C03641=1038.429,245.256,390.466,171.048,41.965,157.999
C03642=1038.436,245.505,390.436,171.051,41.966,157.999
C03643=1038.442,245.753,390.407,171.053,41.968,158.000
C03644=1038.448,246.001,390.378,171.057,41.969,158.001
C03645=1038.454,246.250,390.349,171.059,41.970,158.001
C03646=1038.461,246.497,390.321,171.062,41.972,158.001
C03647=1038.468,246.746,390.291,171.065,41.973,158.002
C03648=1038.474,246.994,390.262,171.068,41.974,158.002
C03649=1038.481,247.242,390.233,171.070,41.976,158.003
C03650=1038.487,247.491,390.204,171.074,41.977,158.003
C03651=1038.494,247.739,390.175,171.077,41.979,158.004
C03652=1038.501,247.987,390.146,171.079,41.980,158.004
C03653=1038.507,248.235,390.117,171.083,41.981,158.005
C03654=1038.515,248.549,390.080,171.085,41.983,158.005
C03655=1038.524,248.863,390.043,171.089,41.985,158.006
C03656=1038.532,249.178,390.007,171.092,41.986,158.006
C03657=1038.541,249.493,389.970,171.096,41.988,158.007
C03658=1038.547,249.741,389.941,171.100,41.989,158.007
C03659=1038.553,249.989,389.912,171.102,41.991,158.008
C03660=1038.560,250.237,389.881,171.105,41.992,158.008
C03661=1038.566,250.485,389.852,171.108,41.994,158.009
C03662=1038.573,250.733,389.823,171.111,41.995,158.009
C03663=1038.579,250.981,389.794,171.114,41.996,158.010
C03664=1038.587,251.230,389.765,171.117,41.998,158.010
C03665=1038.593,251.478,389.736,171.119,41.998,158.011
C03666=1038.600,251.726,389.706,171.123,42.000,158.011
C03667=1038.606,251.974,389.677,171.126,42.001,158.012
C03668=1038.612,252.223,389.648,171.129,42.003,158.012
C03669=1038.619,252.471,389.619,171.132,42.004,158.013
C03670=1038.626,252.719,389.589,171.134,42.005,158.013
C03671=1038.633,252.967,389.561,171.138,42.007,158.014
C03672=1038.640,253.216,389.531,171.140,42.008,158.014
C03673=1038.646,253.463,389.501,171.144,42.009,158.015
C03674=1038.653,253.712,389.472,171.146,42.011,158.015
C03675=1038.659,253.960,389.443,171.149,42.012,158.016
C03676=1038.666,254.208,389.414,171.152,42.013,158.016
C03677=1038.673,254.456,389.384,171.155,42.015,158.016
C03678=1038.679,254.705,389.355,171.159,42.016,158.017
C03679=1038.686,254.953,389.325,171.161,42.018,158.017
C03680=1038.693,255.201,389.296,171.165,42.018,158.018
C03681=1038.700,255.449,389.267,171.167,42.020,158.018
C03682=1038.707,255.697,389.237,171.171,42.021,158.019
C03683=1038.713,255.946,389.208,171.173,42.023,158.019
C03684=1038.720,256.194,389.179,171.176,42.024,158.020
C03685=1038.727,256.442,389.148,171.179,42.025,158.020
C03686=1038.733,256.690,389.119,171.182,42.027,158.021
C03687=1038.740,256.938,389.089,171.186,42.028,158.021
C03688=1038.746,257.187,389.060,171.188,42.029,158.022
C03689=1038.754,257.435,389.030,171.192,42.031,158.022
C03690=1038.761,257.683,389.002,171.194,42.032,158.023
C03691=1038.768,257.931,388.972,171.198,42.033,158.023
C03692=1038.774,258.179,388.943,171.200,42.034,158.024
C03693=1038.781,258.427,388.912,171.204,42.036,158.024
C03694=1038.787,258.675,388.883,171.206,42.037,158.025
C03695=1038.795,258.924,388.853,171.210,42.038,158.025
C03696=1038.801,259.172,388.824,171.212,42.040,158.026
C03697=1038.808,259.420,388.794,171.216,42.041,158.026
C03698=1038.815,259.669,388.765,171.219,42.043,158.027
C03699=1038.821,259.916,388.735,171.222,42.044,158.027
C03700=1038.829,260.164,388.705,171.225,42.045,158.027
C03701=1038.835,260.413,388.676,171.228,42.046,158.028
C03702=1038.843,260.660,388.646,171.232,42.048,158.029
C03703=1038.849,260.909,388.617,171.234,42.049,158.029
C03704=1038.856,261.157,388.587,171.238,42.050,158.029
C03705=1038.863,261.405,388.557,171.240,42.052,158.030
C03706=1038.869,261.653,388.528,171.244,42.053,158.030
C03707=1038.877,261.901,388.498,171.246,42.055,158.031
C03708=1038.884,262.150,388.468,171.250,42.056,158.032
C03709=1038.890,262.397,388.437,171.253,42.058,158.032
C03710=1038.898,262.711,388.400,171.256,42.059,158.033
C03711=1038.906,263.023,388.362,171.261,42.061,158.033
C03712=1038.915,263.336,388.324,171.265,42.063,158.034
C03713=1038.923,263.649,388.287,171.268,42.064,158.034
C03714=1038.930,263.897,388.256,171.272,42.066,158.035
C03715=1038.936,264.145,388.226,171.275,42.067,158.036
C03716=1038.943,264.393,388.196,171.278,42.069,158.036
C03717=1038.950,264.641,388.166,171.281,42.070,158.037
C03718=1038.956,264.889,388.135,171.284,42.072,158.037
C03719=1038.963,265.137,388.105,171.287,42.073,158.038
C03720=1038.971,265.385,388.075,171.291,42.075,158.038
C03721=1038.976,265.633,388.045,171.293,42.076,158.039
C03722=1038.984,265.881,388.015,171.297,42.077,158.039
C03723=1038.991,266.130,387.985,171.300,42.079,158.040
C03724=1038.997,266.378,387.954,171.303,42.080,158.040
C03725=1039.004,266.626,387.924,171.307,42.082,158.041
C03726=1039.011,266.874,387.894,171.309,42.083,158.041
C03727=1039.017,267.122,387.864,171.313,42.085,158.042
C03728=1039.024,267.370,387.834,171.316,42.086,158.042
C03729=1039.031,267.618,387.803,171.319,42.088,158.043
C03730=1039.037,267.866,387.773,171.323,42.089,158.043
C03731=1039.044,268.114,387.743,171.325,42.091,158.044
C03732=1039.050,268.363,387.712,171.329,42.092,158.044
C03733=1039.057,268.610,387.683,171.332,42.093,158.045
C03734=1039.064,268.858,387.651,171.335,42.095,158.045
C03735=1039.071,269.106,387.621,171.339,42.096,158.046
C03736=1039.077,269.354,387.591,171.341,42.098,158.046
C03737=1039.084,269.602,387.560,171.345,42.099,158.047
C03738=1039.090,269.851,387.530,171.348,42.101,158.048
C03739=1039.098,270.099,387.499,171.351,42.102,158.048
C03740=1039.103,270.346,387.469,171.355,42.104,158.049
C03741=1039.111,270.595,387.438,171.357,42.106,158.049
C03742=1039.118,270.843,387.408,171.361,42.107,158.050
C03743=1039.124,271.091,387.377,171.365,42.109,158.050
C03744=1039.131,271.339,387.346,171.367,42.110,158.051
C03745=1039.137,271.587,387.316,171.371,42.111,158.051
C03746=1039.144,271.835,387.285,171.374,42.113,158.052
C03747=1039.151,272.083,387.255,171.377,42.114,158.052
C03748=1039.158,272.331,387.224,171.381,42.116,158.053
C03749=1039.164,272.579,387.193,171.384,42.118,158.054
C03750=1039.171,272.827,387.163,171.387,42.119,158.054
C03751=1039.178,273.075,387.132,171.391,42.121,158.055
C03752=1039.184,273.323,387.101,171.394,42.122,158.055
C03753=1039.191,273.571,387.071,171.397,42.124,158.056
C03754=1039.197,273.819,387.040,171.401,42.125,158.056
C03755=1039.204,274.067,387.009,171.404,42.127,158.057
C03756=1039.211,274.315,386.978,171.407,42.129,158.057
C03757=1039.218,274.563,386.947,171.411,42.130,158.058
C03758=1039.224,274.811,386.916,171.414,42.131,158.059
C03759=1039.231,275.059,386.886,171.417,42.133,158.059
C03760=1039.238,275.307,386.855,171.421,42.135,158.060
C03761=1039.244,275.555,386.824,171.424,42.136,158.060
C03762=1039.252,275.803,386.793,171.427,42.138,158.061
C03763=1039.258,276.051,386.762,171.430,42.139,158.061
C03764=1039.265,276.299,386.731,171.434,42.141,158.062
C03765=1039.272,276.547,386.700,171.437,42.143,158.063
C03766=1039.280,276.864,386.660,171.442,42.145,158.063
C03767=1039.289,277.181,386.620,171.445,42.147,158.064
C03768=1039.297,277.499,386.582,171.450,42.148,158.065
C03769=1039.306,277.816,386.542,171.454,42.150,158.065
C03770=1039.313,278.064,386.510,171.458,42.152,158.066
C03771=1039.320,278.312,386.479,171.461,42.154,158.067
C03772=1039.326,278.560,386.448,171.465,42.155,158.067
C03773=1039.333,278.809,386.417,171.468,42.157,158.068
C03774=1039.340,279.056,386.386,171.471,42.159,158.068
C03775=1039.347,279.304,386.355,171.475,42.160,158.069
C03776=1039.354,279.552,386.323,171.478,42.162,158.069
C03777=1039.360,279.799,386.292,171.481,42.164,158.070
C03778=1039.366,280.048,386.261,171.485,42.165,158.071
C03779=1039.373,280.296,386.230,171.489,42.167,158.071
C03780=1039.380,280.543,386.199,171.491,42.168,158.072
C03781=1039.386,280.791,386.167,171.495,42.170,158.072
C03782=1039.393,281.039,386.136,171.499,42.172,158.073
C03783=1039.400,281.287,386.104,171.502,42.173,158.074
C03784=1039.407,281.535,386.073,171.505,42.175,158.074
C03785=1039.413,281.783,386.041,171.509,42.177,158.075
C03786=1039.420,282.031,386.010,171.513,42.179,158.075
C03787=1039.427,282.279,385.978,171.516,42.180,158.076
C03788=1039.433,282.527,385.947,171.520,42.181,158.076
C03789=1039.440,282.775,385.916,171.523,42.184,158.077
C03790=1039.447,283.022,385.884,171.526,42.185,158.078
C03791=1039.454,283.270,385.853,171.530,42.187,158.078
C03792=1039.460,283.518,385.821,171.534,42.188,158.079
C03793=1039.467,283.766,385.790,171.536,42.190,158.080
C03794=1039.474,284.014,385.758,171.540,42.192,158.080
C03795=1039.481,284.262,385.727,171.544,42.194,158.081
C03796=1039.487,284.510,385.696,171.548,42.195,158.081
C03797=1039.494,284.758,385.664,171.551,42.197,158.082
C03798=1039.501,285.006,385.632,171.555,42.199,158.083
C03799=1039.508,285.254,385.600,171.558,42.200,158.083
C03800=1039.515,285.502,385.569,171.561,42.202,158.084
C03801=1039.522,285.750,385.537,171.565,42.203,158.084
C03802=1039.528,285.997,385.506,171.569,42.205,158.085
C03803=1039.535,286.245,385.474,171.572,42.207,158.086
C03804=1039.542,286.493,385.442,171.576,42.209,158.086
C03805=1039.549,286.740,385.411,171.580,42.210,158.087
C03806=1039.556,286.989,385.379,171.583,42.212,158.087
C03807=1039.562,287.237,385.347,171.586,42.214,158.088
C03808=1039.569,287.485,385.315,171.590,42.216,158.089
C03809=1039.576,287.733,385.284,171.594,42.217,158.089
C03810=1039.583,287.980,385.252,171.597,42.219,158.090
C03811=1039.589,288.228,385.219,171.601,42.221,158.091
C03812=1039.596,288.476,385.188,171.604,42.222,158.091
C03813=1039.603,288.724,385.156,171.608,42.224,158.092
C03814=1039.610,288.972,385.124,171.611,42.226,158.092
C03815=1039.617,289.220,385.093,171.615,42.228,158.093
C03816=1039.623,289.467,385.060,171.619,42.230,158.094
C03817=1039.630,289.715,385.028,171.623,42.231,158.094
C03818=1039.637,289.962,384.996,171.626,42.233,158.095
C03819=1039.644,290.210,384.965,171.630,42.235,158.096
C03820=1039.651,290.459,384.932,171.633,42.237,158.096
C03821=1039.657,290.707,384.900,171.637,42.239,158.097
C03822=1039.666,291.035,384.857,171.642,42.241,158.098
C03823=1039.676,291.365,384.815,171.647,42.243,158.099
C03824=1039.684,291.694,384.772,171.652,42.246,158.099
C03825=1039.693,292.023,384.729,171.657,42.248,158.100
C03826=1039.700,292.271,384.697,171.660,42.250,158.101
C03827=1039.707,292.519,384.665,171.664,42.252,158.102
C03828=1039.713,292.767,384.633,171.668,42.254,158.102
C03829=1039.720,293.015,384.601,171.671,42.255,158.103
C03830=1039.728,293.262,384.569,171.675,42.257,158.104
C03831=1039.734,293.510,384.536,171.678,42.259,158.104
C03832=1039.741,293.757,384.504,171.682,42.261,158.105
C03833=1039.748,294.006,384.472,171.686,42.263,158.106
C03834=1039.755,294.254,384.439,171.689,42.264,158.106
C03835=1039.762,294.501,384.407,171.693,42.266,158.107
C03836=1039.768,294.748,384.374,171.697,42.268,158.107
C03837=1039.775,294.997,384.343,171.701,42.270,158.108
C03838=1039.782,295.245,384.310,171.705,42.272,158.109
C03839=1039.789,295.492,384.278,171.708,42.274,158.109
C03840=1039.796,295.740,384.245,171.712,42.275,158.110
C03841=1039.802,295.988,384.212,171.716,42.277,158.111
C03842=1039.808,296.235,384.179,171.720,42.279,158.112
C03843=1039.815,296.483,384.147,171.723,42.281,158.112
C03844=1039.822,296.731,384.114,171.727,42.283,158.113
C03845=1039.828,296.979,384.081,171.731,42.285,158.114
C03846=1039.835,297.226,384.048,171.735,42.287,158.114
C03847=1039.842,297.474,384.016,171.739,42.289,158.115
C03848=1039.849,297.722,383.983,171.743,42.291,158.116
C03849=1039.855,297.969,383.950,171.746,42.293,158.116
C03850=1039.862,298.218,383.917,171.750,42.295,158.117
C03851=1039.868,298.465,383.885,171.754,42.297,158.118
C03852=1039.875,298.713,383.852,171.758,42.299,158.118
C03853=1039.882,298.961,383.819,171.762,42.301,158.119
C03854=1039.889,299.208,383.786,171.765,42.303,158.120
C03855=1039.896,299.456,383.753,171.769,42.305,158.121
C03856=1039.903,299.703,383.721,171.773,42.307,158.121
C03857=1039.909,299.951,383.688,171.777,42.309,158.122
C03858=1039.916,300.199,383.655,171.781,42.311,158.123
C03859=1039.922,300.447,383.622,171.785,42.313,158.123
C03860=1039.929,300.695,383.588,171.789,42.315,158.124
C03861=1039.936,300.942,383.556,171.792,42.317,158.125
C03862=1039.943,301.189,383.523,171.796,42.319,158.126
C03863=1039.949,301.438,383.490,171.800,42.321,158.126
C03864=1039.956,301.685,383.457,171.804,42.323,158.127
C03865=1039.963,301.933,383.424,171.808,42.325,158.128
C03866=1039.970,302.180,383.391,171.811,42.327,158.128
C03867=1039.977,302.428,383.358,171.815,42.329,158.129
C03868=1039.984,302.675,383.325,171.819,42.331,158.130
C03869=1039.990,302.924,383.292,171.823,42.333,158.131
C03870=1039.997,303.171,383.258,171.827,42.335,158.131
C03871=1040.005,303.419,383.226,171.831,42.337,158.132
C03872=1040.011,303.666,383.193,171.835,42.339,158.133
C03873=1040.018,303.914,383.159,171.838,42.341,158.133
C03874=1040.025,304.162,383.126,171.843,42.343,158.134
C03875=1040.032,304.409,383.093,171.847,42.345,158.135
C03876=1040.039,304.657,383.060,171.851,42.348,158.136
C03877=1040.046,304.904,383.027,171.855,42.350,158.136
C03878=1040.055,305.250,382.980,171.860,42.353,158.137
C03879=1040.065,305.596,382.934,171.866,42.355,158.138
C03880=1040.075,305.942,382.888,171.871,42.358,158.139
C03881=1040.084,306.288,382.841,171.877,42.361,158.140
C03882=1040.091,306.536,382.807,171.882,42.363,158.141
C03883=1040.099,306.783,382.775,171.885,42.365,158.142
C03884=1040.106,307.031,382.741,171.889,42.367,158.143
C03885=1040.113,307.279,382.708,171.893,42.369,158.143
C03886=1040.119,307.526,382.675,171.897,42.371,158.144
C03887=1040.126,307.774,382.641,171.901,42.373,158.145
C03888=1040.133,308.021,382.607,171.905,42.375,158.146
C03889=1040.140,308.270,382.574,171.910,42.377,158.146
C03890=1040.148,308.516,382.541,171.914,42.380,158.147
C03891=1040.155,308.764,382.507,171.917,42.382,158.148
C03892=1040.162,309.012,382.474,171.921,42.384,158.149
C03893=1040.168,309.259,382.441,171.925,42.386,158.149
C03894=1040.176,309.507,382.407,171.930,42.388,158.150
C03895=1040.183,309.755,382.373,171.934,42.390,158.151
C03896=1040.191,310.002,382.340,171.938,42.392,158.152
C03897=1040.197,310.250,382.307,171.942,42.394,158.152
C03898=1040.204,310.497,382.273,171.947,42.396,158.153
C03899=1040.211,310.745,382.240,171.951,42.398,158.154
C03900=1040.219,310.993,382.206,171.955,42.401,158.155
C03901=1040.226,311.240,382.172,171.958,42.403,158.155
C03902=1040.233,311.488,382.138,171.962,42.405,158.156
C03903=1040.240,311.735,382.105,171.967,42.407,158.157
C03904=1040.248,311.982,382.071,171.971,42.409,158.158
C03905=1040.254,312.231,382.038,171.975,42.411,158.159
C03906=1040.261,312.478,382.003,171.979,42.413,158.159
C03907=1040.268,312.726,381.969,171.984,42.416,158.160
C03908=1040.274,312.973,381.935,171.988,42.418,158.161
C03909=1040.281,313.221,381.902,171.992,42.420,158.162
C03910=1040.288,313.469,381.867,171.996,42.423,158.163
C03911=1040.295,313.716,381.833,172.000,42.425,158.163
C03912=1040.301,313.963,381.799,172.005,42.427,158.164
C03913=1040.309,314.211,381.765,172.009,42.430,158.165
C03914=1040.315,314.459,381.730,172.013,42.432,158.166
C03915=1040.322,314.706,381.696,172.017,42.434,158.167
C03916=1040.330,314.953,381.662,172.022,42.436,158.167
C03917=1040.336,315.201,381.628,172.026,42.439,158.168
C03918=1040.343,315.448,381.594,172.030,42.441,158.169
C03919=1040.349,315.696,381.560,172.034,42.443,158.170
C03920=1040.357,315.943,381.525,172.039,42.446,158.171
C03921=1040.363,316.191,381.491,172.043,42.448,158.172
C03922=1040.371,316.438,381.456,172.047,42.451,158.172
C03923=1040.377,316.686,381.422,172.050,42.453,158.173
C03924=1040.384,316.934,381.388,172.056,42.455,158.174
C03925=1040.391,317.181,381.353,172.060,42.458,158.175
C03926=1040.398,317.428,381.319,172.064,42.460,158.176
C03927=1040.404,317.676,381.284,172.068,42.462,158.177
C03928=1040.412,317.923,381.250,172.072,42.464,158.177
C03929=1040.418,318.171,381.216,172.077,42.467,158.178
C03930=1040.426,318.418,381.181,172.082,42.469,158.179
C03931=1040.432,318.666,381.147,172.086,42.472,158.180
C03932=1040.440,318.914,381.112,172.090,42.474,158.181
C03933=1040.446,319.161,381.077,172.093,42.476,158.182
C03934=1040.457,319.512,381.028,172.100,42.480,158.183
C03935=1040.467,319.862,380.980,172.106,42.483,158.184
C03936=1040.477,320.213,380.931,172.113,42.487,158.185
C03937=1040.487,320.563,380.882,172.118,42.490,158.186
C03938=1040.494,320.811,380.847,172.123,42.492,158.187
C03939=1040.501,321.058,380.813,172.127,42.495,158.188
C03940=1040.508,321.306,380.778,172.132,42.497,158.189
C03941=1040.515,321.553,380.743,172.136,42.500,158.190
C03942=1040.522,321.801,380.709,172.141,42.502,158.191
C03943=1040.530,322.049,380.674,172.146,42.505,158.192
C03944=1040.536,322.296,380.639,172.150,42.507,158.193
C03945=1040.543,322.543,380.604,172.155,42.510,158.193
C03946=1040.550,322.791,380.570,172.159,42.512,158.194
C03947=1040.557,323.038,380.535,172.163,42.515,158.195
C03948=1040.565,323.286,380.500,172.168,42.517,158.196
C03949=1040.572,323.533,380.465,172.172,42.519,158.197
C03950=1040.580,323.780,380.430,172.177,42.522,158.198
C03951=1040.586,324.028,380.396,172.181,42.524,158.199
C03952=1040.593,324.276,380.361,172.185,42.527,158.199
C03953=1040.601,324.524,380.326,172.190,42.529,158.200
C03954=1040.608,324.771,380.291,172.194,42.532,158.201
C03955=1040.615,325.018,380.256,172.199,42.534,158.202
C03956=1040.622,325.265,380.221,172.203,42.537,158.203
C03957=1040.630,325.513,380.186,172.208,42.539,158.204
C03958=1040.637,325.760,380.151,172.212,42.541,158.205
C03959=1040.644,326.008,380.117,172.217,42.544,158.206
C03960=1040.652,326.256,380.081,172.222,42.547,158.207
C03961=1040.659,326.503,380.046,172.227,42.549,158.208
C03962=1040.666,326.750,380.011,172.231,42.552,158.208
C03963=1040.674,326.998,379.976,172.236,42.554,158.209
C03964=1040.681,327.245,379.941,172.240,42.557,158.210
C03965=1040.688,327.493,379.906,172.245,42.559,158.211
C03966=1040.696,327.740,379.871,172.249,42.562,158.212
C03967=1040.702,327.988,379.836,172.254,42.564,158.213
C03968=1040.710,328.234,379.801,172.258,42.567,158.214
C03969=1040.718,328.482,379.765,172.263,42.569,158.215
C03970=1040.724,328.729,379.730,172.267,42.572,158.216
C03971=1040.733,328.977,379.695,172.273,42.575,158.217
C03972=1040.740,329.224,379.659,172.277,42.577,158.218
C03973=1040.746,329.471,379.624,172.282,42.580,158.219
C03974=1040.754,329.719,379.589,172.286,42.583,158.219
C03975=1040.761,329.966,379.553,172.291,42.585,158.220
C03976=1040.768,330.214,379.518,172.295,42.588,158.221
C03977=1040.775,330.461,379.482,172.300,42.590,158.222
C03978=1040.782,330.708,379.446,172.306,42.593,158.223
C03979=1040.789,330.956,379.411,172.310,42.596,158.224
C03980=1040.796,331.203,379.375,172.315,42.599,158.225
C03981=1040.804,331.451,379.340,172.319,42.601,158.226
C03982=1040.811,331.698,379.304,172.324,42.604,158.227
C03983=1040.818,331.945,379.269,172.328,42.607,158.228
C03984=1040.825,332.193,379.232,172.334,42.609,158.229
C03985=1040.832,332.440,379.197,172.338,42.613,158.230
C03986=1040.840,332.688,379.161,172.343,42.615,158.231
C03987=1040.847,332.934,379.125,172.348,42.618,158.232
C03988=1040.854,333.182,379.090,172.352,42.620,158.233
C03989=1040.861,333.429,379.054,172.357,42.623,158.234
C03990=1040.871,333.775,379.003,172.364,42.627,158.235
C03991=1040.882,334.121,378.953,172.371,42.631,158.237
C03992=1040.892,334.467,378.904,172.377,42.634,158.238
C03993=1040.902,334.813,378.853,172.384,42.638,158.239
C03994=1040.910,335.060,378.817,172.389,42.641,158.240
C03995=1040.917,335.307,378.781,172.394,42.644,158.241
C03996=1040.925,335.554,378.745,172.399,42.647,158.243
C03997=1040.931,335.802,378.710,172.404,42.650,158.243
C03998=1040.938,336.050,378.673,172.408,42.653,158.244
C03999=1040.946,336.297,378.637,172.413,42.656,158.245
C04000=1040.953,336.544,378.601,172.419,42.659,158.247
C04001=1040.961,336.791,378.565,172.423,42.662,158.248
C04002=1040.967,337.038,378.528,172.428,42.664,158.249
C04003=1040.975,337.286,378.492,172.432,42.667,158.250
C04004=1040.983,337.533,378.456,172.438,42.670,158.251
C04005=1040.989,337.780,378.419,172.443,42.673,158.252
C04006=1040.997,338.028,378.383,172.448,42.676,158.253
C04007=1041.004,338.275,378.347,172.452,42.679,158.254
C04008=1041.011,338.522,378.311,172.458,42.682,158.255
C04009=1041.019,338.769,378.273,172.463,42.685,158.256
C04010=1041.026,339.016,378.237,172.467,42.688,158.257
C04011=1041.034,339.264,378.201,172.473,42.691,158.258
C04012=1041.041,339.511,378.165,172.478,42.693,158.259
C04013=1041.048,339.758,378.128,172.482,42.697,158.260
C04014=1041.056,340.006,378.092,172.487,42.699,158.261
C04015=1041.064,340.253,378.055,172.493,42.702,158.262
C04016=1041.070,340.500,378.019,172.498,42.705,158.263
C04017=1041.078,340.747,377.983,172.502,42.708,158.264
C04018=1041.085,340.995,377.946,172.507,42.711,158.265
C04019=1041.093,341.241,377.909,172.513,42.714,158.266
C04020=1041.100,341.489,377.873,172.518,42.717,158.267
C04021=1041.107,341.736,377.837,172.524,42.720,158.269
C04022=1041.114,341.983,377.799,172.528,42.723,158.270
C04023=1041.122,342.230,377.763,172.533,42.726,158.271
C04024=1041.129,342.478,377.725,172.538,42.729,158.272
C04025=1041.137,342.725,377.689,172.544,42.732,158.273
C04026=1041.144,342.972,377.652,172.548,42.736,158.274
C04027=1041.151,343.219,377.616,172.553,42.739,158.275
C04028=1041.159,343.466,377.578,172.559,42.742,158.276
C04029=1041.166,343.714,377.542,172.564,42.745,158.277
C04030=1041.174,343.961,377.505,172.570,42.748,158.278
C04031=1041.182,344.207,377.468,172.574,42.751,158.279
C04032=1041.188,344.455,377.431,172.579,42.754,158.281
C04033=1041.196,344.702,377.394,172.585,42.757,158.282
C04034=1041.204,344.949,377.356,172.590,42.760,158.283
C04035=1041.211,345.197,377.320,172.595,42.764,158.284
C04036=1041.219,345.444,377.283,172.601,42.767,158.285
C04037=1041.226,345.691,377.245,172.605,42.770,158.286
C04038=1041.234,345.938,377.208,172.610,42.773,158.287
C04039=1041.241,346.185,377.171,172.616,42.777,158.289
C04040=1041.248,346.433,377.134,172.621,42.779,158.290
C04041=1041.256,346.679,377.097,172.627,42.783,158.291
C04042=1041.263,346.927,377.059,172.632,42.786,158.292
C04043=1041.271,347.174,377.022,172.638,42.789,158.293
C04044=1041.278,347.421,376.985,172.642,42.792,158.294
C04045=1041.286,347.668,376.947,172.647,42.796,158.295
C04046=1041.296,348.010,376.896,172.655,42.800,158.297
C04047=1041.306,348.352,376.845,172.662,42.805,158.299
C04048=1041.317,348.694,376.793,172.670,42.809,158.300
C04049=1041.328,349.036,376.741,172.677,42.813,158.302
C04050=1041.335,349.283,376.703,172.683,42.817,158.303
C04051=1041.343,349.530,376.666,172.688,42.820,158.304
C04052=1041.350,349.777,376.629,172.693,42.823,158.305
C04053=1041.357,350.024,376.591,172.699,42.827,158.306
C04054=1041.365,350.272,376.554,172.704,42.830,158.308
C04055=1041.373,350.519,376.516,172.710,42.833,158.309
C04056=1041.380,350.766,376.478,172.715,42.837,158.310
C04057=1041.388,351.013,376.441,172.721,42.840,158.311
C04058=1041.395,351.260,376.403,172.726,42.843,158.312
C04059=1041.403,351.507,376.366,172.732,42.847,158.314
C04060=1041.410,351.754,376.327,172.737,42.850,158.315
C04061=1041.418,352.001,376.289,172.743,42.854,158.316
C04062=1041.425,352.249,376.252,172.748,42.857,158.317
C04063=1041.433,352.495,376.214,172.754,42.860,158.319
C04064=1041.440,352.742,376.176,172.759,42.864,158.320
C04065=1041.448,352.989,376.138,172.765,42.867,158.321
C04066=1041.455,353.237,376.100,172.770,42.871,158.322
C04067=1041.464,353.483,376.062,172.776,42.874,158.324
C04068=1041.471,353.730,376.025,172.781,42.878,158.325
C04069=1041.479,353.977,375.986,172.787,42.881,158.326
C04070=1041.486,354.224,375.949,172.793,42.885,158.327
C04071=1041.494,354.471,375.911,172.798,42.888,158.328
C04072=1041.502,354.719,375.873,172.804,42.891,158.330
C04073=1041.509,354.965,375.834,172.809,42.895,158.331
C04074=1041.517,355.212,375.796,172.815,42.899,158.332
C04075=1041.525,355.459,375.758,172.820,42.902,158.334
C04076=1041.532,355.706,375.720,172.826,42.906,158.335
C04077=1041.540,355.953,375.681,172.831,42.909,158.336
C04078=1041.548,356.200,375.644,172.837,42.913,158.337
C04079=1041.555,356.447,375.606,172.844,42.916,158.339
C04080=1041.563,356.694,375.567,172.849,42.920,158.340
C04081=1041.571,356.941,375.529,172.855,42.923,158.341
C04082=1041.579,357.188,375.490,172.860,42.927,158.343
C04083=1041.587,357.434,375.452,172.866,42.931,158.344
C04084=1041.594,357.681,375.414,172.872,42.934,158.345
C04085=1041.602,357.929,375.376,172.877,42.938,158.346
C04086=1041.609,358.175,375.338,172.883,42.942,158.348
C04087=1041.617,358.423,375.298,172.890,42.945,158.349
C04088=1041.624,358.669,375.260,172.895,42.949,158.350
C04089=1041.633,358.916,375.221,172.901,42.953,158.352
C04090=1041.640,359.163,375.183,172.906,42.956,158.353
C04091=1041.649,359.410,375.144,172.912,42.960,158.354
C04092=1041.656,359.656,375.106,172.919,42.963,158.356
C04093=1041.664,359.903,375.067,172.924,42.967,158.357
C04094=1041.672,360.151,375.028,172.930,42.971,158.358
C04095=1041.679,360.397,374.990,172.936,42.975,158.360
C04096=1041.687,360.645,374.951,172.941,42.978,158.361
C04097=1041.695,360.891,374.913,172.948,42.982,158.362
C04098=1041.703,361.138,374.873,172.954,42.986,158.364
C04099=1041.711,361.385,374.834,172.959,42.990,158.365
C04100=1041.718,361.632,374.796,172.965,42.994,158.366
C04101=1041.727,361.878,374.757,172.972,42.997,158.368
C04102=1041.738,362.226,374.702,172.980,43.003,158.370
C04103=1041.749,362.575,374.647,172.989,43.008,158.372
C04104=1041.759,362.922,374.591,172.997,43.014,158.374
C04105=1041.771,363.271,374.537,173.006,43.019,158.376
C04106=1041.778,363.518,374.497,173.011,43.023,158.377
C04107=1041.786,363.764,374.459,173.017,43.027,158.378
C04108=1041.794,364.011,374.419,173.023,43.031,158.380
C04109=1041.802,364.258,374.380,173.030,43.035,158.381
C04110=1041.809,364.504,374.341,173.035,43.039,158.383
C04111=1041.817,364.751,374.301,173.041,43.043,158.384
C04112=1041.826,364.998,374.263,173.048,43.046,158.385
C04113=1041.833,365.245,374.223,173.054,43.050,158.387
C04114=1041.841,365.491,374.184,173.059,43.054,158.388
C04115=1041.849,365.738,374.144,173.066,43.058,158.390
C04116=1041.857,365.985,374.105,173.072,43.062,158.391
C04117=1041.865,366.232,374.065,173.078,43.066,158.392
C04118=1041.873,366.479,374.026,173.085,43.070,158.394
C04119=1041.880,366.725,373.986,173.091,43.074,158.395
C04120=1041.889,366.971,373.947,173.097,43.078,158.397
C04121=1041.897,367.218,373.907,173.103,43.082,158.398
C04122=1041.905,367.465,373.868,173.109,43.086,158.400
C04123=1041.913,367.712,373.828,173.116,43.090,158.401
C04124=1041.921,367.959,373.789,173.122,43.094,158.403
C04125=1041.929,368.206,373.749,173.128,43.098,158.404
C04126=1041.937,368.452,373.709,173.134,43.103,158.406
C04127=1041.945,368.699,373.669,173.141,43.107,158.407
C04128=1041.954,368.945,373.630,173.147,43.110,158.409
C04129=1041.961,369.192,373.590,173.153,43.115,158.410
C04130=1041.970,369.439,373.551,173.160,43.119,158.412
C04131=1041.977,369.686,373.511,173.166,43.123,158.413
C04132=1041.986,369.933,373.472,173.173,43.127,158.415
C04133=1041.994,370.179,373.432,173.179,43.132,158.416
C04134=1042.002,370.426,373.391,173.185,43.135,158.418
C04135=1042.010,370.672,373.352,173.191,43.140,158.419
C04136=1042.018,370.919,373.312,173.198,43.144,158.421
C04137=1042.026,371.165,373.271,173.204,43.148,158.422
C04138=1042.034,371.412,373.231,173.211,43.153,158.424
C04139=1042.042,371.658,373.191,173.217,43.157,158.425
C04140=1042.050,371.905,373.151,173.224,43.161,158.427
C04141=1042.058,372.152,373.111,173.230,43.165,158.428
C04142=1042.066,372.398,373.071,173.237,43.170,158.430
C04143=1042.074,372.645,373.030,173.244,43.174,158.432
C04144=1042.082,372.892,372.990,173.250,43.179,158.433
C04145=1042.090,373.138,372.950,173.257,43.182,158.435
C04146=1042.099,373.385,372.910,173.263,43.187,158.436
C04147=1042.107,373.632,372.869,173.270,43.191,158.438
C04148=1042.115,373.878,372.829,173.276,43.196,158.439
C04149=1042.122,374.125,372.789,173.283,43.200,158.441
C04150=1042.130,374.371,372.748,173.290,43.204,158.443
C04151=1042.139,374.618,372.707,173.296,43.209,158.444
C04152=1042.148,374.864,372.667,173.303,43.213,158.446
C04153=1042.156,375.111,372.627,173.309,43.218,158.447
C04154=1042.164,375.357,372.587,173.316,43.222,158.449
C04155=1042.172,375.604,372.546,173.323,43.226,158.451
C04156=1042.180,375.850,372.505,173.329,43.231,158.452
C04157=1042.188,376.097,372.464,173.336,43.236,158.454
C04158=1042.201,376.465,372.404,173.346,43.242,158.456
C04159=1042.213,376.832,372.343,173.357,43.249,158.459
C04160=1042.226,377.201,372.282,173.367,43.256,158.461
C04161=1042.238,377.568,372.221,173.377,43.262,158.464
C04162=1042.247,377.815,372.180,173.384,43.267,158.466
C04163=1042.255,378.061,372.140,173.391,43.271,158.467
C04164=1042.263,378.307,372.099,173.397,43.276,158.469
C04165=1042.271,378.554,372.058,173.404,43.280,158.471
C04166=1042.280,378.800,372.017,173.412,43.285,158.472
C04167=1042.288,379.047,371.976,173.419,43.290,158.474
C04168=1042.296,379.293,371.935,173.425,43.295,158.476
C04169=1042.305,379.540,371.893,173.432,43.299,158.477
C04170=1042.313,379.786,371.853,173.439,43.304,158.479
C04171=1042.322,380.033,371.812,173.446,43.309,158.481
C04172=1042.330,380.279,371.770,173.454,43.313,158.483
C04173=1042.338,380.526,371.729,173.460,43.318,158.484
C04174=1042.347,380.771,371.688,173.467,43.323,158.486
C04175=1042.355,381.018,371.647,173.474,43.327,158.488
C04176=1042.363,381.264,371.605,173.481,43.332,158.489
C04177=1042.372,381.511,371.563,173.489,43.337,158.491
C04178=1042.380,381.757,371.522,173.496,43.342,158.493
C04179=1042.389,382.003,371.481,173.502,43.347,158.495
C04180=1042.397,382.249,371.439,173.510,43.352,158.497
C04181=1042.405,382.496,371.398,173.517,43.356,158.498
C04182=1042.414,382.743,371.356,173.524,43.361,158.500
C04183=1042.422,382.988,371.314,173.531,43.366,158.502
C04184=1042.431,383.235,371.273,173.539,43.371,158.504
C04185=1042.439,383.481,371.230,173.546,43.376,158.506
C04186=1042.447,383.728,371.190,173.553,43.381,158.507
C04187=1042.456,383.974,371.148,173.561,43.385,158.509
C04188=1042.465,384.220,371.106,173.568,43.390,158.511
C04189=1042.473,384.466,371.064,173.575,43.395,158.513
C04190=1042.482,384.713,371.023,173.582,43.400,158.515
C04191=1042.491,384.959,370.981,173.590,43.405,158.516
C04192=1042.500,385.206,370.939,173.597,43.410,158.518
C04193=1042.508,385.452,370.897,173.605,43.415,158.520
C04194=1042.516,385.698,370.856,173.612,43.420,158.522
C04195=1042.525,385.944,370.814,173.619,43.425,158.524
C04196=1042.534,386.190,370.771,173.627,43.430,158.526
C04197=1042.542,386.437,370.729,173.634,43.435,158.528
C04198=1042.551,386.683,370.687,173.642,43.440,158.529
C04199=1042.560,386.929,370.646,173.649,43.445,158.531
C04200=1042.569,387.176,370.603,173.656,43.450,158.533
C04201=1042.578,387.422,370.561,173.664,43.455,158.535
C04202=1042.587,387.668,370.519,173.671,43.460,158.537
C04203=1042.596,387.915,370.478,173.679,43.465,158.539
C04204=1042.604,388.161,370.435,173.686,43.471,158.541
C04205=1042.613,388.407,370.393,173.693,43.476,158.543
C04206=1042.621,388.652,370.350,173.701,43.481,158.545
C04207=1042.630,388.899,370.308,173.710,43.486,158.547
C04208=1042.638,389.145,370.265,173.717,43.491,158.548
C04209=1042.647,389.391,370.224,173.724,43.496,158.550
C04210=1042.656,389.637,370.181,173.732,43.502,158.552
C04211=1042.665,389.883,370.138,173.740,43.507,158.554
C04212=1042.674,390.130,370.096,173.747,43.512,158.556
C04213=1042.683,390.376,370.053,173.756,43.518,158.558
C04214=1042.697,390.778,369.983,173.768,43.526,158.562
C04215=1042.711,391.179,369.913,173.781,43.535,158.565
C04216=1042.726,391.581,369.844,173.793,43.544,158.568
C04217=1042.740,391.983,369.774,173.806,43.552,158.571
C04218=1042.749,392.229,369.731,173.814,43.558,158.573
C04219=1042.758,392.474,369.689,173.822,43.564,158.575
C04220=1042.766,392.720,369.646,173.830,43.569,158.577
C04221=1042.776,392.967,369.602,173.838,43.574,158.579
C04222=1042.784,393.213,369.559,173.846,43.579,158.581
C04223=1042.794,393.458,369.516,173.853,43.585,158.584
C04224=1042.802,393.704,369.473,173.862,43.591,158.586
C04225=1042.811,393.951,369.430,173.870,43.596,158.588
C04226=1042.820,394.197,369.387,173.877,43.602,158.590
C04227=1042.829,394.442,369.344,173.886,43.607,158.592
C04228=1042.838,394.688,369.301,173.894,43.613,158.594
C04229=1042.847,394.935,369.257,173.903,43.618,158.596
C04230=1042.856,395.180,369.214,173.910,43.624,158.598
C04231=1042.866,395.427,369.171,173.918,43.630,158.600
C04232=1042.874,395.673,369.127,173.927,43.635,158.602
C04233=1042.883,395.919,369.084,173.935,43.641,158.605
C04234=1042.892,396.165,369.040,173.943,43.646,158.607
C04235=1042.901,396.411,368.997,173.951,43.652,158.609
C04236=1042.910,396.657,368.953,173.960,43.658,158.611
C04237=1042.920,396.902,368.909,173.968,43.664,158.613
C04238=1042.929,397.149,368.866,173.976,43.670,158.615
C04239=1042.938,397.394,368.822,173.984,43.675,158.618
C04240=1042.946,397.640,368.779,173.992,43.681,158.620
C04241=1042.956,397.886,368.735,174.001,43.687,158.622
C04242=1042.965,398.133,368.691,174.009,43.693,158.624
C04243=1042.974,398.378,368.647,174.018,43.698,158.626
C04244=1042.983,398.624,368.603,174.027,43.704,158.628
C04245=1042.992,398.870,368.559,174.034,43.710,158.631
C04246=1043.001,399.116,368.515,174.044,43.716,158.633
C04247=1043.011,399.362,368.471,174.051,43.722,158.635
C04248=1043.020,399.607,368.427,174.060,43.728,158.637
C04249=1043.029,399.853,368.383,174.069,43.734,158.640
C04250=1043.038,400.099,368.339,174.077,43.740,158.642
C04251=1043.047,400.345,368.296,174.086,43.745,158.644
C04252=1043.057,400.591,368.251,174.094,43.752,158.646
C04253=1043.066,400.837,368.207,174.103,43.757,158.649
C04254=1043.076,401.083,368.162,174.112,43.764,158.651
C04255=1043.085,401.328,368.119,174.120,43.769,158.653
C04256=1043.094,401.574,368.075,174.129,43.776,158.656
C04257=1043.103,401.820,368.031,174.138,43.782,158.658
C04258=1043.113,402.066,367.986,174.146,43.788,158.660
C04259=1043.122,402.312,367.941,174.155,43.794,158.663
C04260=1043.131,402.558,367.896,174.164,43.800,158.665
C04261=1043.140,402.803,367.852,174.173,43.806,158.667
C04262=1043.150,403.049,367.808,174.181,43.812,158.670
C04263=1043.159,403.295,367.764,174.191,43.819,158.672
C04264=1043.168,403.541,367.718,174.200,43.825,158.674
C04265=1043.178,403.786,367.673,174.209,43.831,158.677
C04266=1043.188,404.032,367.629,174.218,43.837,158.679
C04267=1043.197,404.278,367.584,174.226,43.844,158.682
C04268=1043.206,404.524,367.539,174.235,43.850,158.684
C04269=1043.216,404.769,367.494,174.244,43.856,158.686
C04270=1043.229,405.112,367.431,174.257,43.865,158.690
C04271=1043.242,405.454,367.368,174.269,43.874,158.693
C04272=1043.256,405.797,367.306,174.283,43.882,158.697
C04273=1043.268,406.139,367.243,174.295,43.892,158.700
C04274=1043.278,406.384,367.199,174.305,43.898,158.703
C04275=1043.287,406.631,367.153,174.314,43.904,158.705
C04276=1043.297,406.876,367.108,174.323,43.911,158.708
C04277=1043.306,407.122,367.062,174.333,43.917,158.710
C04278=1043.316,407.367,367.017,174.342,43.924,158.713
C04279=1043.326,407.613,366.972,174.351,43.930,158.715
C04280=1043.335,407.859,366.926,174.360,43.937,158.718
C04281=1043.345,408.104,366.881,174.370,43.943,158.720
C04282=1043.354,408.350,366.835,174.379,43.950,158.723
C04283=1043.365,408.596,366.790,174.389,43.957,158.725
C04284=1043.374,408.841,366.744,174.398,43.963,158.728
C04285=1043.384,409.087,366.699,174.407,43.970,158.730
C04286=1043.394,409.332,366.653,174.417,43.976,158.733
C04287=1043.403,409.578,366.608,174.426,43.983,158.736
C04288=1043.414,409.824,366.562,174.436,43.990,158.738
C04289=1043.423,410.070,366.517,174.445,43.997,158.741
C04290=1043.434,410.315,366.471,174.456,44.003,158.743
C04291=1043.443,410.560,366.425,174.465,44.010,158.746
C04292=1043.453,410.807,366.379,174.474,44.016,158.749
C04293=1043.462,411.052,366.333,174.484,44.024,158.751
C04294=1043.473,411.297,366.287,174.495,44.030,158.754
C04295=1043.482,411.543,366.241,174.504,44.037,158.757
C04296=1043.493,411.789,366.196,174.514,44.044,158.759
C04297=1043.503,412.034,366.150,174.523,44.050,158.762
C04298=1043.513,412.280,366.104,174.534,44.057,158.765
C04299=1043.522,412.526,366.057,174.543,44.064,158.767
C04300=1043.532,412.771,366.011,174.553,44.071,158.770
C04301=1043.543,413.016,365.965,174.564,44.078,158.773
C04302=1043.555,413.340,365.903,174.577,44.088,158.777
C04303=1043.568,413.665,365.842,174.589,44.097,158.780
C04304=1043.581,413.989,365.781,174.603,44.106,158.784
C04305=1043.595,414.312,365.719,174.616,44.116,158.788
C04306=1043.605,414.558,365.673,174.627,44.123,158.790
C04307=1043.615,414.804,365.627,174.637,44.130,158.793
C04308=1043.625,415.049,365.580,174.647,44.137,158.796
C04309=1043.635,415.294,365.534,174.657,44.144,158.799
C04310=1043.645,415.540,365.486,174.668,44.151,158.802
C04311=1043.655,415.785,365.439,174.678,44.158,158.805
C04312=1043.666,416.031,365.393,174.688,44.165,158.807
C04313=1043.676,416.276,365.346,174.698,44.173,158.810
C04314=1043.686,416.521,365.299,174.709,44.180,158.813
C04315=1043.696,416.767,365.252,174.719,44.188,158.816
C04316=1043.706,417.012,365.205,174.730,44.194,158.819
C04317=1043.717,417.257,365.158,174.741,44.202,158.822
C04318=1043.727,417.503,365.111,174.751,44.209,158.825
C04319=1043.737,417.748,365.064,174.762,44.216,158.828
C04320=1043.748,417.993,365.017,174.773,44.224,158.831
C04321=1043.758,418.238,364.970,174.783,44.232,158.834
C04322=1043.769,418.484,364.922,174.793,44.238,158.836
C04323=1043.779,418.730,364.875,174.804,44.246,158.839
C04324=1043.789,418.975,364.828,174.815,44.254,158.843
C04325=1043.799,419.220,364.780,174.826,44.261,158.846
C04326=1043.808,419.434,364.739,174.835,44.268,158.848
C04327=1043.817,419.648,364.698,174.845,44.274,158.851
C04328=1043.827,419.863,364.656,174.854,44.281,158.854
C04329=1043.835,420.078,364.614,174.864,44.287,158.856
C04330=1043.844,420.292,364.572,174.873,44.295,158.859
C04331=1043.854,420.507,364.531,174.883,44.301,158.862
C04332=1043.863,420.720,364.489,174.892,44.307,158.864
C04333=1043.872,420.935,364.447,174.902,44.315,158.867
C04334=1043.883,421.181,364.399,174.913,44.322,158.870
C04335=1043.893,421.425,364.351,174.925,44.330,158.873
C04336=1043.904,421.670,364.303,174.936,44.337,158.876
C04337=1043.914,421.916,364.256,174.947,44.345,158.879
C04338=1043.925,422.161,364.208,174.958,44.353,158.883
C04339=1043.936,422.406,364.160,174.970,44.361,158.886
C04340=1043.946,422.651,364.111,174.981,44.368,158.889
C04341=1043.956,422.897,364.064,174.992,44.376,158.892
C04342=1043.967,423.142,364.016,175.003,44.384,158.895
C04343=1043.978,423.387,363.967,175.015,44.392,158.898
C04344=1043.989,423.632,363.919,175.026,44.400,158.902
C04345=1044.000,423.877,363.871,175.037,44.408,158.905
C04346=1044.010,424.122,363.823,175.050,44.416,158.908
C04347=1044.021,424.367,363.774,175.061,44.424,158.912
C04348=1044.032,424.612,363.725,175.072,44.432,158.915
C04349=1044.043,424.857,363.677,175.084,44.440,158.918
C04350=1044.053,425.102,363.629,175.095,44.448,158.921
C04351=1044.064,425.347,363.579,175.108,44.456,158.925
C04352=1044.075,425.593,363.531,175.119,44.464,158.928
C04353=1044.086,425.837,363.482,175.131,44.472,158.931
C04354=1044.096,426.082,363.434,175.143,44.481,158.935
C04355=1044.108,426.327,363.385,175.155,44.489,158.938
C04356=1044.119,426.572,363.336,175.166,44.497,158.941
C04357=1044.130,426.817,363.287,175.179,44.505,158.945
C04358=1044.140,427.061,363.238,175.191,44.513,158.948
C04359=1044.151,427.307,363.189,175.202,44.522,158.952
C04360=1044.162,427.552,363.140,175.215,44.530,158.955
C04361=1044.174,427.797,363.091,175.227,44.539,158.959
C04362=1044.184,428.042,363.041,175.240,44.547,158.962
C04363=1044.196,428.286,362.992,175.251,44.555,158.966
C04364=1044.206,428.531,362.943,175.264,44.563,158.969
C04365=1044.218,428.777,362.893,175.276,44.572,158.973
C04366=1044.229,429.022,362.844,175.288,44.580,158.976
C04367=1044.240,429.267,362.795,175.301,44.589,158.980
C04368=1044.251,429.512,362.745,175.313,44.598,158.983
C04369=1044.263,429.756,362.696,175.326,44.606,158.987
C04370=1044.273,430.001,362.646,175.338,44.615,158.990
C04371=1044.284,430.246,362.596,175.351,44.623,158.994
C04372=1044.296,430.490,362.547,175.364,44.632,158.998
C04373=1044.306,430.735,362.497,175.377,44.641,159.001
C04374=1044.317,430.980,362.447,175.389,44.649,159.005
C04375=1044.330,431.224,362.397,175.401,44.658,159.009
C04376=1044.340,431.469,362.347,175.414,44.667,159.012
C04377=1044.352,431.714,362.297,175.428,44.676,159.016
C04378=1044.364,431.959,362.247,175.441,44.684,159.020
C04379=1044.374,432.204,362.197,175.453,44.693,159.023
C04380=1044.386,432.448,362.147,175.466,44.702,159.027
C04381=1044.398,432.693,362.097,175.479,44.711,159.031
C04382=1044.409,432.937,362.046,175.492,44.720,159.035
C04383=1044.421,433.182,361.996,175.505,44.729,159.038
C04384=1044.432,433.427,361.946,175.518,44.738,159.042
C04385=1044.444,433.672,361.895,175.532,44.747,159.046
C04386=1044.455,433.896,361.849,175.544,44.755,159.049
C04387=1044.465,434.121,361.803,175.556,44.763,159.053
C04388=1044.476,434.345,361.756,175.569,44.771,159.057
C04389=1044.486,434.570,361.710,175.581,44.780,159.060
C04390=1044.498,434.794,361.664,175.594,44.788,159.064
C04391=1044.508,435.018,361.617,175.605,44.796,159.067
C04392=1044.519,435.244,361.570,175.618,44.805,159.071
C04393=1044.530,435.468,361.524,175.631,44.814,159.074
C04394=1044.542,435.712,361.473,175.644,44.823,159.078
C04395=1044.553,435.957,361.422,175.658,44.832,159.082
C04396=1044.565,436.201,361.371,175.672,44.841,159.086
C04397=1044.577,436.445,361.320,175.685,44.850,159.090
C04398=1044.589,436.690,361.269,175.700,44.860,159.094
C04399=1044.601,436.935,361.218,175.713,44.869,159.098
C04400=1044.612,437.179,361.167,175.727,44.878,159.102
C04401=1044.624,437.423,361.116,175.741,44.888,159.106
C04402=1044.636,437.668,361.064,175.755,44.897,159.110
C04403=1044.647,437.912,361.013,175.770,44.907,159.115
C04404=1044.660,438.156,360.961,175.783,44.916,159.119
C04405=1044.672,438.401,360.909,175.798,44.926,159.123
C04406=1044.683,438.645,360.858,175.812,44.935,159.127
C04407=1044.696,438.890,360.807,175.826,44.945,159.131
C04408=1044.708,439.133,360.755,175.841,44.954,159.135
C04409=1044.720,439.378,360.703,175.855,44.964,159.140
C04410=1044.732,439.622,360.651,175.870,44.974,159.144
C04411=1044.745,439.867,360.600,175.885,44.984,159.148
C04412=1044.757,440.111,360.547,175.898,44.993,159.152
C04413=1044.769,440.355,360.496,175.913,45.003,159.157
C04414=1044.781,440.599,360.444,175.928,45.013,159.161
C04415=1044.794,440.844,360.391,175.943,45.022,159.165
C04416=1044.806,441.088,360.339,175.958,45.033,159.170
C04417=1044.817,441.332,360.287,175.973,45.042,159.174
C04418=1044.830,441.577,360.234,175.988,45.052,159.178
C04419=1044.842,441.820,360.182,176.002,45.062,159.183
C04420=1044.855,442.064,360.130,176.017,45.072,159.187
C04421=1044.867,442.309,360.077,176.033,45.082,159.192
C04422=1044.880,442.553,360.025,176.049,45.092,159.196
C04423=1044.892,442.797,359.973,176.064,45.102,159.201
C04424=1044.905,443.041,359.920,176.079,45.112,159.205
C04425=1044.917,443.286,359.867,176.094,45.122,159.209
C04426=1044.929,443.529,359.814,176.109,45.132,159.214
C04427=1044.942,443.773,359.762,176.125,45.143,159.219
C04428=1044.955,444.017,359.708,176.140,45.153,159.223
C04429=1044.968,444.261,359.656,176.157,45.163,159.228
C04430=1044.981,444.505,359.603,176.172,45.174,159.232
C04431=1044.994,444.749,359.550,176.187,45.184,159.237
C04432=1045.006,444.993,359.497,176.204,45.194,159.242
C04433=1045.018,445.237,359.444,176.219,45.204,159.246
C04434=1045.032,445.480,359.391,176.236,45.215,159.251
C04435=1045.046,445.722,359.339,176.251,45.225,159.255
C04436=1045.060,445.966,359.288,176.267,45.235,159.260
C04437=1045.075,446.210,359.236,176.284,45.245,159.265
C04438=1045.091,446.454,359.186,176.300,45.255,159.269
C04439=1045.107,446.698,359.135,176.316,45.264,159.274
C04440=1045.124,446.942,359.085,176.333,45.274,159.278
C04441=1045.141,447.186,359.036,176.349,45.284,159.283
C04442=1045.160,447.430,358.987,176.365,45.293,159.287
C04443=1045.179,447.673,358.939,176.382,45.302,159.292
C04444=1045.198,447.919,358.890,176.399,45.311,159.296
C04445=1045.218,448.163,358.844,176.415,45.320,159.300
C04446=1045.238,448.402,358.798,176.432,45.328,159.305
C04447=1045.259,448.642,358.752,176.449,45.337,159.309
C04448=1045.281,448.881,358.708,176.466,45.346,159.313
C04449=1045.303,449.120,358.663,176.482,45.354,159.318
C04450=1045.325,449.359,358.619,176.499,45.362,159.322
C04451=1045.349,449.599,358.576,176.516,45.370,159.326
C04452=1045.373,449.839,358.534,176.532,45.378,159.330
C04453=1045.397,450.078,358.491,176.550,45.386,159.334
C04454=1045.423,450.323,358.448,176.567,45.394,159.338
C04455=1045.450,450.569,358.406,176.584,45.401,159.343
C04456=1045.476,450.815,358.364,176.602,45.409,159.347
C04457=1045.503,451.060,358.322,176.619,45.417,159.351
C04458=1045.199,451.097,358.012,176.621,45.500,159.376
C04459=1045.172,450.851,358.054,176.604,45.493,159.372
C04460=1045.144,450.606,358.096,176.586,45.485,159.368
C04461=1045.118,450.361,358.138,176.568,45.477,159.363
C04462=1045.092,450.115,358.181,176.551,45.470,159.359
C04463=1045.067,449.884,358.221,176.534,45.462,159.355
C04464=1045.044,449.653,358.263,176.518,45.455,159.351
C04465=1045.022,449.422,358.305,176.502,45.447,159.347
C04466=1045.000,449.191,358.347,176.485,45.439,159.343
C04467=1044.978,448.960,358.390,176.470,45.431,159.339
C04468=1044.957,448.729,358.433,176.453,45.423,159.335
C04469=1044.937,448.497,358.476,176.437,45.415,159.331
C04470=1044.917,448.267,358.520,176.421,45.407,159.327
C04471=1044.896,448.022,358.568,176.404,45.398,159.322
C04472=1044.877,447.777,358.615,176.388,45.389,159.318
C04473=1044.857,447.533,358.662,176.370,45.380,159.313
C04474=1044.839,447.289,358.712,176.354,45.371,159.309
C04475=1044.821,447.045,358.761,176.337,45.361,159.304
C04476=1044.803,446.801,358.810,176.321,45.352,159.300
C04477=1044.787,446.558,358.860,176.305,45.342,159.295
C04478=1044.771,446.313,358.911,176.289,45.333,159.291
C04479=1044.756,446.070,358.961,176.272,45.323,159.286
C04480=1044.740,445.825,359.013,176.256,45.314,159.282
C04481=1044.727,445.583,359.065,176.239,45.303,159.277
C04482=1044.712,445.341,359.117,176.224,45.293,159.272
C04483=1044.699,445.097,359.170,176.207,45.283,159.268
C04484=1044.686,444.853,359.224,176.192,45.273,159.263
C04485=1044.674,444.609,359.276,176.176,45.263,159.259
C04486=1044.661,444.365,359.329,176.160,45.252,159.254
C04487=1044.649,444.121,359.382,176.145,45.242,159.249
C04488=1044.636,443.877,359.435,176.128,45.232,159.245
C04489=1044.623,443.633,359.488,176.113,45.222,159.240
C04490=1044.611,443.389,359.541,176.098,45.212,159.236
C04491=1044.598,443.145,359.593,176.082,45.202,159.231
C04492=1044.586,442.901,359.646,176.067,45.192,159.227
C04493=1044.573,442.657,359.699,176.051,45.182,159.222
C04494=1044.561,442.413,359.751,176.036,45.172,159.218
C04495=1044.548,442.169,359.804,176.021,45.162,159.213
C04496=1044.536,441.925,359.857,176.005,45.152,159.209
C04497=1044.523,441.680,359.909,175.990,45.142,159.204
C04498=1044.511,441.436,359.961,175.975,45.132,159.200
C04499=1044.499,441.192,360.013,175.960,45.122,159.196
C04500=1044.486,440.948,360.066,175.945,45.112,159.191
C04501=1044.474,440.704,360.118,175.930,45.103,159.187
C04502=1044.462,440.459,360.169,175.916,45.093,159.183
C04503=1044.449,440.215,360.222,175.901,45.083,159.178
C04504=1044.437,439.971,360.274,175.887,45.074,159.174
C04505=1044.425,439.726,360.325,175.872,45.064,159.170
C04506=1044.413,439.483,360.378,175.857,45.054,159.166
C04507=1044.401,439.238,360.429,175.843,45.045,159.161
C04508=1044.389,438.994,360.481,175.828,45.035,159.157
C04509=1044.376,438.749,360.533,175.813,45.026,159.153
C04510=1044.365,438.504,360.584,175.800,45.016,159.149
C04511=1044.352,438.261,360.636,175.785,45.007,159.145
C04512=1044.340,438.016,360.688,175.771,44.997,159.141
C04513=1044.328,437.772,360.739,175.757,44.988,159.136
C04514=1044.316,437.527,360.790,175.743,44.979,159.132
C04515=1044.305,437.284,360.841,175.728,44.969,159.128
C04516=1044.293,437.039,360.892,175.715,44.960,159.124
C04517=1044.281,436.795,360.944,175.700,44.950,159.120
C04518=1044.269,436.550,360.995,175.687,44.941,159.116
C04519=1044.257,436.306,361.047,175.672,44.932,159.112
C04520=1044.245,436.061,361.097,175.659,44.923,159.108
C04521=1044.234,435.817,361.148,175.645,44.914,159.104
C04522=1044.222,435.572,361.199,175.631,44.905,159.100
C04523=1044.211,435.347,361.246,175.619,44.896,159.097
C04524=1044.199,435.121,361.293,175.606,44.888,159.093
C04525=1044.189,434.896,361.340,175.594,44.880,159.089
C04526=1044.178,434.670,361.386,175.581,44.871,159.086
C04527=1044.167,434.444,361.433,175.568,44.863,159.082
C04528=1044.157,434.219,361.479,175.556,44.854,159.079
C04529=1044.146,433.994,361.526,175.543,44.846,159.075
C04530=1044.135,433.768,361.573,175.532,44.838,159.072
C04531=1044.123,433.523,361.623,175.518,44.829,159.068
C04532=1044.112,433.279,361.673,175.505,44.820,159.064
C04533=1044.100,433.034,361.724,175.492,44.811,159.060
C04534=1044.089,432.790,361.774,175.479,44.802,159.056
C04535=1044.077,432.545,361.825,175.466,44.794,159.053
C04536=1044.065,432.301,361.874,175.452,44.785,159.049
C04537=1044.054,432.056,361.925,175.439,44.776,159.045
C04538=1044.043,431.810,361.975,175.426,44.768,159.041
C04539=1044.031,431.566,362.024,175.413,44.759,159.038
C04540=1044.020,431.322,362.075,175.400,44.750,159.034
C04541=1044.009,431.076,362.125,175.387,44.741,159.030
C04542=1043.997,430.832,362.174,175.375,44.733,159.027
C04543=1043.986,430.587,362.225,175.362,44.724,159.023
C04544=1043.975,430.343,362.274,175.349,44.715,159.019
C04545=1043.964,430.098,362.324,175.336,44.707,159.016
C04546=1043.953,429.853,362.374,175.325,44.698,159.012
C04547=1043.941,429.608,362.423,175.312,44.690,159.009
C04548=1043.930,429.363,362.473,175.299,44.682,159.005
C04549=1043.919,429.119,362.522,175.287,44.673,159.001
C04550=1043.908,428.874,362.572,175.274,44.665,158.998
C04551=1043.898,428.629,362.622,175.261,44.656,158.994
C04552=1043.886,428.384,362.671,175.250,44.648,158.991
C04553=1043.875,428.139,362.720,175.237,44.640,158.987
C04554=1043.864,427.894,362.769,175.225,44.631,158.984
C04555=1043.853,427.649,362.818,175.212,44.623,158.980
C04556=1043.842,427.404,362.868,175.201,44.614,158.977
C04557=1043.831,427.159,362.917,175.188,44.606,158.974
C04558=1043.820,426.914,362.965,175.176,44.598,158.970
C04559=1043.809,426.669,363.015,175.164,44.590,158.967
C04560=1043.798,426.424,363.064,175.152,44.582,158.963
C04561=1043.786,426.179,363.112,175.141,44.574,158.960
C04562=1043.776,425.935,363.161,175.128,44.565,158.957
C04563=1043.765,425.690,363.210,175.117,44.558,158.953
C04564=1043.754,425.444,363.259,175.105,44.549,158.950
C04565=1043.743,425.199,363.307,175.093,44.542,158.947
C04566=1043.733,424.955,363.356,175.081,44.533,158.943
C04567=1043.722,424.709,363.404,175.070,44.525,158.940
C04568=1043.711,424.464,363.453,175.058,44.517,158.937
C04569=1043.700,424.220,363.502,175.046,44.509,158.933
C04570=1043.689,423.974,363.550,175.034,44.501,158.930
C04571=1043.678,423.729,363.599,175.023,44.494,158.927
C04572=1043.668,423.484,363.646,175.011,44.486,158.924
C04573=1043.657,423.239,363.695,175.000,44.478,158.920
C04574=1043.646,422.994,363.743,174.989,44.470,158.917
C04575=1043.635,422.749,363.791,174.976,44.462,158.914
C04576=1043.625,422.503,363.840,174.965,44.455,158.911
C04577=1043.614,422.258,363.887,174.954,44.447,158.908
C04578=1043.604,422.013,363.935,174.943,44.439,158.904
C04579=1043.593,421.768,363.983,174.931,44.431,158.901
C04580=1043.582,421.523,364.031,174.920,44.424,158.898
C04581=1043.572,421.277,364.079,174.909,44.416,158.895
C04582=1043.561,421.033,364.127,174.898,44.409,158.892
C04583=1043.552,420.818,364.169,174.888,44.402,158.889
C04584=1043.543,420.601,364.211,174.878,44.395,158.887
C04585=1043.534,420.386,364.253,174.869,44.389,158.884
C04586=1043.524,420.171,364.295,174.859,44.382,158.881
C04587=1043.515,419.955,364.336,174.850,44.375,158.878
C04588=1043.506,419.740,364.378,174.840,44.369,158.876
C04589=1043.496,419.524,364.420,174.830,44.362,158.873
C04590=1043.488,419.309,364.463,174.821,44.356,158.870
C04591=1043.478,419.063,364.510,174.810,44.348,158.867
C04592=1043.468,418.818,364.557,174.799,44.341,158.864
C04593=1043.457,418.573,364.604,174.789,44.333,158.861
C04594=1043.447,418.328,364.651,174.778,44.326,158.858
C04595=1043.437,418.082,364.699,174.767,44.318,158.855
C04596=1043.426,417.837,364.745,174.756,44.311,158.852
C04597=1043.415,417.591,364.793,174.746,44.304,158.850
C04598=1043.405,417.346,364.840,174.735,44.296,158.847
C04599=1043.395,417.101,364.887,174.724,44.289,158.844
C04600=1043.385,416.855,364.935,174.714,44.282,158.841
C04601=1043.374,416.610,364.982,174.703,44.275,158.838
C04602=1043.364,416.365,365.028,174.692,44.267,158.835
C04603=1043.354,416.119,365.075,174.683,44.260,158.832
C04604=1043.343,415.874,365.122,174.672,44.253,158.829
C04605=1043.334,415.628,365.169,174.662,44.246,158.826
C04606=1043.323,415.383,365.216,174.651,44.239,158.824
C04607=1043.313,415.139,365.262,174.641,44.232,158.821
C04608=1043.303,414.893,365.309,174.630,44.225,158.818
C04609=1043.293,414.647,365.356,174.621,44.218,158.815
C04610=1043.283,414.401,365.402,174.610,44.211,158.812
C04611=1043.272,414.156,365.448,174.600,44.204,158.810
C04612=1043.263,413.911,365.495,174.590,44.197,158.807
C04613=1043.253,413.665,365.542,174.580,44.190,158.804
C04614=1043.243,413.419,365.588,174.569,44.183,158.801
C04615=1043.233,413.174,365.635,174.559,44.175,158.798
C04616=1043.223,412.929,365.681,174.550,44.169,158.796
C04617=1043.213,412.683,365.727,174.539,44.162,158.793
C04618=1043.203,412.437,365.774,174.529,44.155,158.790
C04619=1043.194,412.192,365.820,174.520,44.148,158.787
C04620=1043.183,411.947,365.866,174.509,44.141,158.785
C04621=1043.173,411.701,365.912,174.500,44.135,158.782
C04622=1043.163,411.456,365.958,174.490,44.128,158.779
C04623=1043.154,411.209,366.004,174.480,44.121,158.777
C04624=1043.144,410.964,366.049,174.470,44.114,158.774
C04625=1043.133,410.719,366.095,174.461,44.108,158.771
C04626=1043.123,410.473,366.142,174.451,44.101,158.769
C04627=1043.113,410.227,366.186,174.440,44.094,158.766
C04628=1043.104,409.982,366.233,174.431,44.087,158.763
C04629=1043.094,409.737,366.278,174.422,44.081,158.761
C04630=1043.084,409.490,366.324,174.412,44.074,158.758
C04631=1043.074,409.245,366.370,174.403,44.068,158.756
C04632=1043.065,408.999,366.415,174.393,44.061,158.753
C04633=1043.054,408.754,366.461,174.384,44.055,158.751
C04634=1043.045,408.508,366.506,174.374,44.048,158.748
C04635=1043.036,408.262,366.551,174.364,44.042,158.745
C04636=1043.025,408.017,366.597,174.355,44.035,158.743
C04637=1043.016,407.771,366.643,174.346,44.029,158.740
C04638=1043.006,407.526,366.687,174.336,44.022,158.738
C04639=1042.996,407.280,366.733,174.327,44.016,158.735
C04640=1042.987,407.034,366.779,174.318,44.009,158.733
C04641=1042.977,406.789,366.824,174.308,44.003,158.730
C04642=1042.968,406.543,366.869,174.299,43.997,158.728
C04643=1042.960,406.331,366.908,174.291,43.991,158.726
C04644=1042.951,406.119,366.946,174.283,43.986,158.724
C04645=1042.943,405.909,366.985,174.275,43.980,158.721
C04646=1042.935,405.696,367.024,174.268,43.975,158.719
C04647=1042.927,405.485,367.063,174.260,43.969,158.717
C04648=1042.919,405.274,367.102,174.251,43.964,158.715
C04649=1042.911,405.062,367.141,174.243,43.958,158.713
C04650=1042.902,404.850,367.179,174.236,43.953,158.711
C04651=1042.894,404.633,367.220,174.228,43.947,158.709
C04652=1042.886,404.415,367.259,174.220,43.942,158.707
C04653=1042.877,404.198,367.299,174.212,43.936,158.704
C04654=1042.869,403.980,367.338,174.204,43.930,158.702
C04655=1042.860,403.763,367.378,174.195,43.925,158.700
C04656=1042.853,403.545,367.418,174.188,43.920,158.698
C04657=1042.845,403.327,367.457,174.180,43.914,158.696
C04658=1042.836,403.110,367.497,174.172,43.909,158.694
C04659=1042.827,402.864,367.541,174.163,43.903,158.692
C04660=1042.817,402.618,367.586,174.154,43.897,158.689
C04661=1042.807,402.372,367.630,174.146,43.890,158.687
C04662=1042.798,402.127,367.675,174.137,43.885,158.685
C04663=1042.790,401.881,367.720,174.128,43.879,158.682
C04664=1042.780,401.635,367.764,174.119,43.872,158.680
C04665=1042.770,401.389,367.809,174.111,43.867,158.678
C04666=1042.761,401.143,367.853,174.102,43.860,158.675
C04667=1042.752,400.897,367.897,174.093,43.855,158.673
C04668=1042.743,400.652,367.941,174.085,43.848,158.671
C04669=1042.733,400.406,367.985,174.076,43.843,158.668
C04670=1042.724,400.160,368.029,174.067,43.837,158.666
C04671=1042.715,399.914,368.073,174.059,43.831,158.664
C04672=1042.706,399.668,368.117,174.050,43.825,158.662
C04673=1042.696,399.422,368.161,174.041,43.820,158.659
C04674=1042.687,399.177,368.205,174.033,43.813,158.657
C04675=1042.678,398.931,368.249,174.024,43.807,158.655
C04676=1042.668,398.684,368.293,174.016,43.802,158.653
C04677=1042.660,398.439,368.337,174.007,43.796,158.650
C04678=1042.650,398.193,368.381,173.998,43.790,158.648
C04679=1042.641,397.947,368.425,173.990,43.785,158.646
C04680=1042.632,397.701,368.469,173.982,43.779,158.644
C04681=1042.622,397.455,368.512,173.974,43.773,158.642
C04682=1042.613,397.209,368.556,173.965,43.767,158.639
C04683=1042.604,396.963,368.600,173.957,43.761,158.637
C04684=1042.595,396.717,368.643,173.948,43.756,158.635
C04685=1042.587,396.472,368.686,173.940,43.750,158.633
C04686=1042.577,396.226,368.731,173.932,43.745,158.631
C04687=1042.569,395.980,368.774,173.924,43.739,158.629
C04688=1042.559,395.733,368.818,173.915,43.733,158.626
C04689=1042.551,395.487,368.861,173.907,43.728,158.624
C04690=1042.541,395.242,368.904,173.899,43.722,158.622
C04691=1042.532,394.996,368.947,173.891,43.716,158.620
C04692=1042.523,394.750,368.991,173.883,43.711,158.618
C04693=1042.514,394.503,369.034,173.874,43.705,158.616
C04694=1042.505,394.258,369.077,173.867,43.700,158.614
C04695=1042.496,394.012,369.121,173.859,43.695,158.612
C04696=1042.487,393.765,369.164,173.850,43.689,158.610
C04697=1042.478,393.520,369.206,173.842,43.684,158.608
C04698=1042.469,393.274,369.249,173.834,43.678,158.605
C04699=1042.461,393.028,369.292,173.826,43.673,158.603
C04700=1042.451,392.781,369.335,173.818,43.667,158.601
C04701=1042.442,392.536,369.379,173.810,43.662,158.599
C04702=1042.434,392.290,369.422,173.802,43.657,158.597
C04703=1042.426,392.059,369.461,173.795,43.652,158.595
C04704=1042.417,391.829,369.502,173.787,43.647,158.594
C04705=1042.409,391.599,369.542,173.780,43.642,158.592
C04706=1042.401,391.369,369.582,173.772,43.637,158.590
C04707=1042.393,391.139,369.622,173.766,43.632,158.588
C04708=1042.385,390.909,369.661,173.758,43.626,158.586
C04709=1042.376,390.679,369.702,173.751,43.622,158.584
C04710=1042.368,390.449,369.742,173.744,43.617,158.582
C04711=1042.359,390.203,369.784,173.736,43.612,158.580
C04712=1042.351,389.956,369.827,173.728,43.606,158.578
C04713=1042.341,389.711,369.869,173.720,43.601,158.576
C04714=1042.333,389.464,369.912,173.713,43.596,158.575
C04715=1042.324,389.218,369.954,173.705,43.591,158.573
C04716=1042.315,388.972,369.997,173.697,43.586,158.571
C04717=1042.306,388.726,370.039,173.690,43.580,158.569
C04718=1042.298,388.480,370.082,173.682,43.576,158.567
C04719=1042.289,388.234,370.124,173.674,43.570,158.565
C04720=1042.281,387.987,370.166,173.667,43.565,158.563
C04721=1042.272,387.741,370.208,173.659,43.560,158.561
C04722=1042.262,387.495,370.251,173.652,43.555,158.559
C04723=1042.253,387.249,370.292,173.644,43.550,158.557
C04724=1042.245,387.002,370.335,173.637,43.545,158.555
C04725=1042.236,386.756,370.376,173.629,43.540,158.554
C04726=1042.227,386.510,370.419,173.621,43.535,158.552
C04727=1042.219,386.263,370.461,173.614,43.530,158.550
C04728=1042.210,386.017,370.503,173.606,43.525,158.548
C04729=1042.201,385.771,370.545,173.599,43.520,158.546
C04730=1042.193,385.525,370.586,173.591,43.515,158.544
C04731=1042.184,385.278,370.628,173.584,43.510,158.542
C04732=1042.176,385.032,370.670,173.577,43.506,158.541
C04733=1042.167,384.785,370.712,173.569,43.501,158.539
C04734=1042.157,384.540,370.754,173.562,43.495,158.537
C04735=1042.150,384.293,370.795,173.555,43.491,158.535
C04736=1042.141,384.047,370.837,173.547,43.486,158.533
C04737=1042.132,383.800,370.879,173.540,43.481,158.531
C04738=1042.124,383.555,370.920,173.533,43.476,158.530
C04739=1042.116,383.308,370.962,173.525,43.471,158.528
C04740=1042.107,383.062,371.004,173.518,43.466,158.526
C04741=1042.098,382.815,371.046,173.511,43.462,158.524
C04742=1042.090,382.569,371.086,173.503,43.457,158.522
C04743=1042.081,382.323,371.128,173.497,43.452,158.521
C04744=1042.073,382.077,371.170,173.490,43.448,158.519
C04745=1042.064,381.830,371.212,173.483,43.443,158.517
C04746=1042.056,381.583,371.253,173.475,43.438,158.515
C04747=1042.047,381.338,371.294,173.468,43.433,158.514
C04748=1042.039,381.091,371.336,173.461,43.429,158.512
C04749=1042.031,380.845,371.377,173.454,43.424,158.510
C04750=1042.022,380.598,371.419,173.446,43.419,158.508
C04751=1042.014,380.352,371.459,173.440,43.415,158.507
C04752=1042.005,380.106,371.501,173.433,43.410,158.505
C04753=1041.998,379.859,371.542,173.426,43.405,158.503
C04754=1041.989,379.613,371.584,173.419,43.401,158.501
C04755=1041.981,379.367,371.625,173.411,43.396,158.500
C04756=1041.972,379.120,371.666,173.405,43.391,158.498
C04757=1041.964,378.874,371.707,173.398,43.386,158.496
C04758=1041.956,378.628,371.748,173.391,43.382,158.495
C04759=1041.947,378.381,371.789,173.384,43.378,158.493
C04760=1041.939,378.134,371.829,173.378,43.373,158.491
C04761=1041.931,377.887,371.870,173.370,43.368,158.490
C04762=1041.922,377.642,371.912,173.363,43.364,158.488
C04763=1041.910,377.272,371.972,173.353,43.357,158.485
C04764=1041.897,376.901,372.034,173.343,43.350,158.483
C04765=1041.885,376.531,372.095,173.333,43.344,158.480
C04766=1041.872,376.162,372.155,173.323,43.337,158.478
C04767=1041.864,375.915,372.196,173.316,43.333,158.476
C04768=1041.855,375.668,372.237,173.309,43.328,158.475
C04769=1041.847,375.422,372.278,173.301,43.324,158.473
C04770=1041.839,375.176,372.318,173.295,43.319,158.471
C04771=1041.831,374.929,372.359,173.288,43.315,158.470
C04772=1041.823,374.682,372.400,173.282,43.311,158.468
C04773=1041.814,374.436,372.439,173.275,43.306,158.467
C04774=1041.806,374.190,372.480,173.268,43.302,158.465
C04775=1041.798,373.943,372.520,173.262,43.298,158.464
C04776=1041.790,373.697,372.561,173.255,43.294,158.462
C04777=1041.782,373.449,372.601,173.248,43.289,158.460
C04778=1041.774,373.203,372.642,173.242,43.285,158.459
C04779=1041.765,372.957,372.682,173.235,43.281,158.457
C04780=1041.757,372.710,372.722,173.229,43.276,158.456
C04781=1041.749,372.464,372.763,173.222,43.272,158.454
C04782=1041.742,372.217,372.803,173.215,43.268,158.452
C04783=1041.734,371.971,372.843,173.209,43.264,158.451
C04784=1041.726,371.724,372.883,173.202,43.259,158.449
C04785=1041.717,371.478,372.923,173.196,43.255,158.448
C04786=1041.709,371.231,372.963,173.189,43.251,158.446
C04787=1041.701,370.985,373.004,173.184,43.247,158.445
C04788=1041.693,370.737,373.044,173.177,43.243,158.443
C04789=1041.685,370.490,373.084,173.171,43.238,158.442
C04790=1041.676,370.244,373.124,173.164,43.234,158.440
C04791=1041.669,369.997,373.164,173.158,43.230,158.439
C04792=1041.660,369.751,373.203,173.151,43.226,158.437
C04793=1041.653,369.504,373.243,173.145,43.222,158.436
C04794=1041.644,369.257,373.282,173.138,43.218,158.434
C04795=1041.636,369.010,373.322,173.132,43.214,158.433
C04796=1041.628,368.764,373.362,173.125,43.210,158.431
C04797=1041.620,368.517,373.402,173.119,43.206,158.430
C04798=1041.611,368.271,373.442,173.113,43.202,158.428
C04799=1041.604,368.024,373.482,173.107,43.198,158.427
C04800=1041.595,367.777,373.521,173.100,43.194,158.425
C04801=1041.588,367.531,373.560,173.094,43.190,158.424
C04802=1041.580,367.285,373.600,173.088,43.186,158.422
C04803=1041.572,367.038,373.640,173.081,43.182,158.421
C04804=1041.564,366.790,373.678,173.076,43.178,158.419
C04805=1041.556,366.543,373.718,173.069,43.174,158.418
C04806=1041.548,366.297,373.757,173.063,43.170,158.417
C04807=1041.540,366.050,373.797,173.056,43.166,158.415
C04808=1041.532,365.804,373.836,173.050,43.162,158.414
C04809=1041.524,365.557,373.876,173.044,43.158,158.412
C04810=1041.516,365.310,373.915,173.038,43.154,158.411
C04811=1041.508,365.063,373.955,173.032,43.150,158.409
C04812=1041.500,364.816,373.994,173.026,43.146,158.408
C04813=1041.493,364.570,374.034,173.019,43.142,158.406
C04814=1041.485,364.323,374.072,173.013,43.138,158.405
C04815=1041.476,364.076,374.112,173.008,43.135,158.404
C04816=1041.469,363.830,374.150,173.001,43.131,158.402
C04817=1041.461,363.583,374.190,172.995,43.127,158.401
C04818=1041.453,363.336,374.230,172.990,43.123,158.400
C04819=1041.442,362.986,374.285,172.981,43.118,158.398
C04820=1041.432,362.636,374.340,172.973,43.112,158.396
C04821=1041.420,362.286,374.396,172.964,43.107,158.394
C04822=1041.409,361.936,374.451,172.955,43.102,158.392
C04823=1041.401,361.689,374.489,172.949,43.098,158.390
C04824=1041.393,361.442,374.529,172.943,43.094,158.389
C04825=1041.386,361.195,374.567,172.938,43.090,158.388
C04826=1041.378,360.948,374.606,172.931,43.087,158.386
C04827=1041.370,360.702,374.645,172.925,43.083,158.385
C04828=1041.362,360.455,374.684,172.920,43.079,158.383
C04829=1041.354,360.207,374.723,172.914,43.075,158.382
C04830=1041.347,359.961,374.761,172.907,43.072,158.381
C04831=1041.339,359.714,374.800,172.901,43.068,158.379
C04832=1041.331,359.467,374.838,172.896,43.065,158.378
C04833=1041.323,359.220,374.877,172.890,43.061,158.377
C04834=1041.315,358.973,374.915,172.885,43.057,158.376
C04835=1041.308,358.727,374.955,172.878,43.054,158.374
C04836=1041.300,358.480,374.993,172.872,43.050,158.373
C04837=1041.292,358.233,375.032,172.867,43.047,158.372
C04838=1041.284,357.986,375.070,172.861,43.043,158.370
C04839=1041.277,357.738,375.108,172.855,43.039,158.369
C04840=1041.269,357.492,375.146,172.850,43.036,158.368
C04841=1041.261,357.245,375.185,172.843,43.033,158.366
C04842=1041.253,356.998,375.223,172.838,43.029,158.365
C04843=1041.246,356.751,375.262,172.832,43.025,158.364
C04844=1041.238,356.504,375.300,172.826,43.022,158.363
C04845=1041.231,356.258,375.338,172.821,43.018,158.361
C04846=1041.223,356.010,375.376,172.815,43.015,158.360
C04847=1041.215,355.764,375.414,172.810,43.011,158.359
C04848=1041.206,355.516,375.453,172.803,43.008,158.357
C04849=1041.199,355.269,375.490,172.797,43.004,158.356
C04850=1041.192,355.023,375.528,172.792,43.001,158.355
C04851=1041.184,354.776,375.567,172.786,42.997,158.354
C04852=1041.176,354.528,375.604,172.781,42.994,158.352
C04853=1041.169,354.282,375.643,172.775,42.991,158.351
C04854=1041.161,354.035,375.681,172.770,42.987,158.350
C04855=1041.153,353.788,375.719,172.764,42.984,158.349
C04856=1041.146,353.541,375.757,172.759,42.980,158.347
C04857=1041.138,353.293,375.795,172.753,42.977,158.346
C04858=1041.130,353.047,375.833,172.748,42.973,158.345
C04859=1041.123,352.800,375.871,172.742,42.970,158.344
C04860=1041.115,352.553,375.908,172.737,42.966,158.343
C04861=1041.107,352.306,375.946,172.731,42.963,158.341
C04862=1041.100,352.058,375.984,172.725,42.960,158.340
C04863=1041.092,351.812,376.022,172.720,42.957,158.339
C04864=1041.085,351.565,376.060,172.715,42.953,158.338
C04865=1041.078,351.318,376.097,172.709,42.950,158.337
C04866=1041.070,351.070,376.136,172.704,42.946,158.335
C04867=1041.062,350.823,376.173,172.698,42.943,158.334
C04868=1041.055,350.576,376.211,172.693,42.940,158.333
C04869=1041.047,350.329,376.248,172.687,42.937,158.332
C04870=1041.040,350.083,376.286,172.682,42.933,158.331
C04871=1041.032,349.836,376.324,172.676,42.930,158.329
C04872=1041.024,349.588,376.361,172.671,42.927,158.328
C04873=1041.016,349.341,376.398,172.665,42.924,158.327
C04874=1041.009,349.094,376.436,172.660,42.920,158.326
C04875=1040.999,348.750,376.488,172.652,42.916,158.324
C04876=1040.988,348.405,376.540,172.645,42.911,158.323
C04877=1040.978,348.062,376.593,172.637,42.907,158.321
C04878=1040.967,347.718,376.644,172.630,42.903,158.319
C04879=1040.960,347.470,376.681,172.624,42.899,158.318
C04880=1040.953,347.223,376.719,172.619,42.896,158.317
C04881=1040.945,346.976,376.756,172.614,42.893,158.316
C04882=1040.937,346.729,376.793,172.608,42.890,158.315
C04883=1040.930,346.482,376.831,172.603,42.886,158.314
C04884=1040.922,346.235,376.867,172.597,42.884,158.312
C04885=1040.915,345.988,376.904,172.592,42.881,158.311
C04886=1040.907,345.741,376.941,172.588,42.877,158.310
C04887=1040.900,345.494,376.979,172.582,42.874,158.309
C04888=1040.893,345.247,377.016,172.577,42.871,158.308
C04889=1040.885,344.999,377.053,172.571,42.868,158.307
C04890=1040.878,344.752,377.090,172.566,42.865,158.306
C04891=1040.870,344.505,377.127,172.561,42.862,158.305
C04892=1040.863,344.257,377.164,172.555,42.859,158.303
C04893=1040.855,344.011,377.201,172.551,42.856,158.302
C04894=1040.848,343.763,377.238,172.546,42.853,158.301
C04895=1040.841,343.516,377.275,172.540,42.849,158.300
C04896=1040.833,343.269,377.312,172.535,42.846,158.299
C04897=1040.826,343.022,377.349,172.530,42.843,158.298
C04898=1040.818,342.775,377.385,172.525,42.840,158.297
C04899=1040.812,342.527,377.422,172.520,42.838,158.296
C04900=1040.804,342.280,377.459,172.515,42.834,158.295
C04901=1040.797,342.033,377.496,172.509,42.831,158.294
C04902=1040.789,341.786,377.533,172.504,42.828,158.292
C04903=1040.782,341.539,377.569,172.500,42.825,158.291
C04904=1040.775,341.291,377.606,172.494,42.822,158.290
C04905=1040.767,341.044,377.643,172.489,42.819,158.289
C04906=1040.759,340.797,377.679,172.484,42.817,158.288
C04907=1040.752,340.549,377.716,172.478,42.814,158.287
C04908=1040.744,340.302,377.752,172.474,42.811,158.286
C04909=1040.737,340.056,377.788,172.469,42.808,158.285
C04910=1040.730,339.808,377.825,172.464,42.805,158.284
C04911=1040.722,339.560,377.861,172.458,42.802,158.283
C04912=1040.715,339.313,377.898,172.454,42.799,158.282
C04913=1040.708,339.066,377.933,172.449,42.796,158.281
C04914=1040.700,338.819,377.971,172.443,42.793,158.280
C04915=1040.693,338.572,378.007,172.438,42.790,158.279
C04916=1040.685,338.324,378.043,172.434,42.788,158.278
C04917=1040.678,338.078,378.079,172.429,42.785,158.277
C04918=1040.671,337.830,378.116,172.423,42.782,158.276
C04919=1040.663,337.582,378.152,172.419,42.779,158.275
C04920=1040.656,337.336,378.188,172.414,42.776,158.274
C04921=1040.649,337.088,378.225,172.409,42.773,158.273
C04922=1040.642,336.840,378.261,172.405,42.771,158.272
C04923=1040.635,336.594,378.297,172.399,42.768,158.271
C04924=1040.627,336.346,378.333,172.394,42.765,158.270
C04925=1040.621,336.099,378.370,172.390,42.762,158.269
C04926=1040.613,335.852,378.406,172.384,42.759,158.267
C04927=1040.605,335.604,378.442,172.379,42.757,158.267
C04928=1040.598,335.357,378.478,172.375,42.753,158.266
C04929=1040.591,335.109,378.513,172.370,42.751,158.264
C04930=1040.584,334.863,378.549,172.365,42.748,158.264
C04931=1040.573,334.514,378.601,172.358,42.744,158.262
C04932=1040.563,334.166,378.651,172.351,42.740,158.261
C04933=1040.553,333.819,378.701,172.344,42.736,158.259
C04934=1040.543,333.471,378.751,172.338,42.733,158.258
C04935=1040.535,333.224,378.787,172.333,42.730,158.257
C04936=1040.528,332.977,378.823,172.328,42.727,158.256
C04937=1040.520,332.729,378.859,172.323,42.725,158.255
C04938=1040.513,332.482,378.895,172.318,42.722,158.254
C04939=1040.506,332.234,378.930,172.314,42.719,158.253
C04940=1040.499,331.987,378.966,172.309,42.717,158.252
C04941=1040.491,331.740,379.002,172.305,42.714,158.251
C04942=1040.484,331.493,379.037,172.299,42.711,158.250
C04943=1040.477,331.246,379.073,172.294,42.709,158.249
C04944=1040.470,330.998,379.109,172.290,42.706,158.248
C04945=1040.463,330.751,379.145,172.285,42.703,158.247
C04946=1040.456,330.503,379.180,172.281,42.701,158.246
C04947=1040.449,330.256,379.215,172.276,42.698,158.245
C04948=1040.441,330.008,379.251,172.272,42.695,158.245
C04949=1040.434,329.761,379.287,172.266,42.693,158.244
C04950=1040.427,329.514,379.322,172.262,42.690,158.243
C04951=1040.420,329.266,379.358,172.257,42.688,158.242
C04952=1040.413,329.019,379.393,172.253,42.685,158.241
C04953=1040.406,328.772,379.429,172.248,42.682,158.240
C04954=1040.398,328.524,379.464,172.243,42.680,158.239
C04955=1040.391,328.277,379.499,172.239,42.678,158.238
C04956=1040.384,328.029,379.534,172.234,42.675,158.237
C04957=1040.376,327.782,379.569,172.229,42.672,158.236
C04958=1040.370,327.534,379.604,172.224,42.670,158.235
C04959=1040.361,327.287,379.640,172.220,42.667,158.234
C04960=1040.354,327.040,379.675,172.215,42.665,158.233
C04961=1040.347,326.793,379.709,172.211,42.662,158.233
C04962=1040.339,326.545,379.745,172.206,42.660,158.232
C04963=1040.333,326.297,379.780,172.202,42.658,158.231
C04964=1040.325,326.050,379.815,172.197,42.655,158.230
C04965=1040.318,325.802,379.850,172.193,42.653,158.229
C04966=1040.310,325.555,379.885,172.188,42.650,158.228
C04967=1040.304,325.308,379.920,172.184,42.648,158.227
C04968=1040.295,325.060,379.955,172.179,42.646,158.226
C04969=1040.289,324.813,379.990,172.175,42.643,158.226
C04970=1040.281,324.566,380.024,172.170,42.641,158.225
C04971=1040.274,324.318,380.059,172.165,42.638,158.224
C04972=1040.267,324.070,380.094,172.160,42.636,158.223
C04973=1040.260,323.823,380.129,172.156,42.633,158.222
C04974=1040.253,323.575,380.164,172.151,42.631,158.221
C04975=1040.246,323.328,380.198,172.147,42.629,158.220
C04976=1040.239,323.081,380.234,172.142,42.626,158.219
C04977=1040.231,322.833,380.268,172.138,42.624,158.218
C04978=1040.224,322.585,380.303,172.134,42.621,158.218
C04979=1040.217,322.338,380.337,172.129,42.619,158.217
C04980=1040.210,322.091,380.373,172.125,42.616,158.216
C04981=1040.202,321.844,380.407,172.120,42.614,158.215
C04982=1040.196,321.596,380.442,172.116,42.611,158.214
C04983=1040.188,321.348,380.476,172.111,42.610,158.213
C04984=1040.181,321.100,380.512,172.107,42.607,158.212
C04985=1040.174,320.853,380.545,172.103,42.605,158.212
C04986=1040.167,320.605,380.581,172.098,42.602,158.211
C04987=1040.157,320.253,380.630,172.091,42.599,158.209
C04988=1040.147,319.900,380.679,172.086,42.595,158.208
C04989=1040.137,319.548,380.728,172.079,42.592,158.207
C04990=1040.127,319.195,380.777,172.073,42.589,158.206
C04991=1040.120,318.948,380.812,172.069,42.587,158.205
C04992=1040.113,318.700,380.847,172.064,42.584,158.204
C04993=1040.106,318.453,380.881,172.060,42.582,158.203
C04994=1040.099,318.205,380.916,172.056,42.579,158.202
C04995=1040.092,317.958,380.950,172.051,42.578,158.202
C04996=1040.085,317.710,380.984,172.047,42.575,158.201
C04997=1040.078,317.463,381.019,172.043,42.573,158.200
C04998=1040.071,317.216,381.052,172.038,42.570,158.199
C04999=1040.065,316.968,381.087,172.034,42.568,158.198
C05000=1040.057,316.721,381.121,172.030,42.566,158.198
C05001=1040.051,316.473,381.156,172.026,42.563,158.197
C05002=1040.043,316.226,381.190,172.021,42.561,158.196
C05003=1040.037,315.978,381.225,172.017,42.559,158.195
C05004=1040.029,315.731,381.259,172.013,42.556,158.194
C05005=1040.023,315.483,381.294,172.008,42.555,158.193
C05006=1040.016,315.235,381.327,172.004,42.552,158.193
C05007=1040.010,314.988,381.362,172.000,42.550,158.192
C05008=1040.002,314.741,381.396,171.996,42.548,158.191
C05009=1039.996,314.493,381.430,171.991,42.545,158.190
C05010=1039.989,314.245,381.464,171.987,42.543,158.189
C05011=1039.981,313.998,381.499,171.983,42.541,158.189
C05012=1039.975,313.750,381.533,171.979,42.538,158.188
C05013=1039.968,313.503,381.567,171.974,42.537,158.187
C05014=1039.962,313.255,381.601,171.970,42.534,158.186
C05015=1039.954,313.007,381.635,171.966,42.532,158.185
C05016=1039.948,312.759,381.669,171.962,42.530,158.185
C05017=1039.941,312.513,381.703,171.957,42.527,158.184
C05018=1039.935,312.265,381.738,171.954,42.525,158.183
C05019=1039.927,312.017,381.772,171.950,42.523,158.182
C05020=1039.920,311.770,381.806,171.946,42.521,158.181
C05021=1039.913,311.522,381.839,171.941,42.519,158.181
C05022=1039.906,311.275,381.872,171.937,42.517,158.180
C05023=1039.899,311.027,381.905,171.933,42.515,158.179
C05024=1039.892,310.779,381.939,171.929,42.513,158.178
C05025=1039.884,310.532,381.973,171.924,42.511,158.178
C05026=1039.877,310.284,382.007,171.920,42.508,158.177
C05027=1039.870,310.036,382.041,171.916,42.506,158.176
C05028=1039.864,309.789,382.073,171.913,42.504,158.175
C05029=1039.856,309.541,382.107,171.908,42.503,158.175
C05030=1039.849,309.294,382.140,171.904,42.500,158.174
C05031=1039.841,309.046,382.174,171.900,42.498,158.173
C05032=1039.835,308.798,382.207,171.896,42.496,158.172
C05033=1039.828,308.551,382.241,171.892,42.494,158.172
C05034=1039.821,308.303,382.275,171.887,42.492,158.171
C05035=1039.814,308.056,382.308,171.883,42.490,158.170
C05036=1039.806,307.808,382.341,171.879,42.488,158.169
C05037=1039.799,307.560,382.374,171.876,42.486,158.169
C05038=1039.793,307.313,382.408,171.872,42.484,158.168
C05039=1039.786,307.065,382.441,171.867,42.482,158.167
C05040=1039.779,306.817,382.475,171.863,42.480,158.166
C05041=1039.772,306.570,382.508,171.859,42.478,158.166
C05042=1039.764,306.323,382.541,171.855,42.476,158.165
C05043=1039.755,305.974,382.588,171.849,42.473,158.164
C05044=1039.745,305.627,382.634,171.844,42.470,158.163
C05045=1039.735,305.279,382.682,171.839,42.468,158.162
C05046=1039.726,304.931,382.728,171.832,42.465,158.161
C05047=1039.719,304.683,382.761,171.829,42.463,158.160
C05048=1039.711,304.436,382.794,171.825,42.461,158.159
C05049=1039.704,304.188,382.827,171.821,42.459,158.159
C05050=1039.698,303.941,382.861,171.817,42.457,158.158
C05051=1039.691,303.693,382.894,171.813,42.455,158.157
C05052=1039.684,303.445,382.927,171.808,42.453,158.156
C05053=1039.677,303.198,382.960,171.804,42.451,158.156
C05054=1039.670,302.950,382.993,171.801,42.449,158.155
C05055=1039.663,302.703,383.026,171.797,42.447,158.154
C05056=1039.656,302.454,383.059,171.793,42.445,158.154
C05057=1039.650,302.207,383.092,171.789,42.443,158.153
C05058=1039.643,301.959,383.126,171.785,42.441,158.152
C05059=1039.636,301.712,383.158,171.781,42.439,158.152
C05060=1039.630,301.464,383.191,171.778,42.437,158.151
C05061=1039.623,301.216,383.224,171.774,42.435,158.150
C05062=1039.616,300.969,383.257,171.770,42.433,158.149
C05063=1039.608,300.721,383.290,171.766,42.431,158.149
C05064=1039.602,300.473,383.323,171.761,42.430,158.148
C05065=1039.595,300.225,383.356,171.757,42.428,158.147
C05066=1039.589,299.978,383.389,171.754,42.426,158.147
C05067=1039.582,299.730,383.422,171.750,42.424,158.146
C05068=1039.575,299.483,383.454,171.746,42.422,158.145
C05069=1039.568,299.235,383.487,171.742,42.420,158.145
C05070=1039.561,298.987,383.520,171.738,42.418,158.144
C05071=1039.555,298.739,383.553,171.734,42.416,158.143
C05072=1039.548,298.492,383.585,171.731,42.414,158.142
C05073=1039.541,298.244,383.619,171.727,42.412,158.142
C05074=1039.535,297.997,383.652,171.723,42.410,158.141
C05075=1039.528,297.749,383.685,171.719,42.408,158.140
C05076=1039.521,297.501,383.718,171.715,42.406,158.140
C05077=1039.514,297.253,383.750,171.712,42.405,158.139
C05078=1039.508,297.006,383.783,171.708,42.403,158.138
C05079=1039.501,296.757,383.816,171.704,42.401,158.138
C05080=1039.495,296.510,383.848,171.700,42.399,158.137
C05081=1039.488,296.263,383.881,171.696,42.397,158.136
C05082=1039.481,296.014,383.914,171.693,42.395,158.136
C05083=1039.475,295.767,383.946,171.689,42.393,158.135
C05084=1039.468,295.519,383.979,171.686,42.391,158.134
C05085=1039.461,295.272,384.011,171.682,42.389,158.133
C05086=1039.455,295.023,384.044,171.679,42.388,158.133
C05087=1039.448,294.776,384.076,171.675,42.386,158.132
C05088=1039.442,294.528,384.109,171.671,42.384,158.132
C05089=1039.434,294.280,384.141,171.667,42.382,158.131
C05090=1039.427,294.032,384.173,171.663,42.381,158.130
C05091=1039.421,293.785,384.205,171.660,42.379,158.130
C05092=1039.413,293.537,384.238,171.656,42.377,158.129
C05093=1039.407,293.289,384.271,171.652,42.375,158.128
C05094=1039.400,293.041,384.302,171.648,42.373,158.128
C05095=1039.393,292.794,384.334,171.644,42.371,158.127
C05096=1039.386,292.546,384.367,171.641,42.370,158.126
C05097=1039.380,292.298,384.399,171.637,42.368,158.126
C05098=1039.373,292.050,384.431,171.633,42.366,158.125
C05099=1039.364,291.719,384.474,171.628,42.364,158.124
C05100=1039.355,291.388,384.517,171.623,42.362,158.123
C05101=1039.345,291.057,384.560,171.618,42.359,158.123
C05102=1039.336,290.725,384.603,171.613,42.357,158.122
C05103=1039.330,290.477,384.635,171.610,42.356,158.121
C05104=1039.322,290.230,384.667,171.607,42.354,158.120
C05105=1039.316,289.982,384.699,171.603,42.352,158.120
C05106=1039.309,289.735,384.731,171.599,42.350,158.119
C05107=1039.302,289.486,384.763,171.596,42.348,158.118
C05108=1039.296,289.238,384.795,171.592,42.347,158.118
C05109=1039.289,288.991,384.827,171.588,42.345,158.117
C05110=1039.282,288.743,384.858,171.585,42.344,158.117
C05111=1039.275,288.495,384.890,171.581,42.342,158.116
C05112=1039.269,288.247,384.922,171.577,42.340,158.115
C05113=1039.262,287.999,384.955,171.573,42.338,158.115
C05114=1039.255,287.751,384.986,171.571,42.337,158.114
C05115=1039.248,287.503,385.018,171.567,42.335,158.114
C05116=1039.241,287.256,385.050,171.563,42.333,158.113
C05117=1039.235,287.008,385.081,171.559,42.331,158.112
C05118=1039.229,286.760,385.113,171.556,42.330,158.112
C05119=1039.222,286.512,385.145,171.552,42.328,158.111
C05120=1039.214,286.264,385.177,171.548,42.327,158.111
C05121=1039.207,286.016,385.209,171.545,42.325,158.110
C05122=1039.201,285.768,385.240,171.542,42.323,158.109
C05123=1039.194,285.520,385.272,171.538,42.322,158.109
C05124=1039.187,285.272,385.303,171.534,42.320,158.108
C05125=1039.181,285.025,385.335,171.531,42.319,158.108
C05126=1039.174,284.777,385.367,171.527,42.317,158.107
C05127=1039.167,284.529,385.398,171.523,42.315,158.106
C05128=1039.160,284.282,385.430,171.520,42.314,158.106
C05129=1039.153,284.034,385.461,171.517,42.312,158.105
C05130=1039.147,283.786,385.492,171.513,42.310,158.105
C05131=1039.140,283.538,385.524,171.510,42.309,158.104
C05132=1039.133,283.289,385.556,171.506,42.307,158.103
C05133=1039.126,283.041,385.587,171.502,42.306,158.103
C05134=1039.119,282.793,385.618,171.500,42.304,158.102
C05135=1039.112,282.545,385.650,171.496,42.302,158.102
C05136=1039.106,282.298,385.681,171.492,42.301,158.101
C05137=1039.099,282.050,385.713,171.489,42.299,158.100
C05138=1039.092,281.802,385.744,171.485,42.297,158.100
C05139=1039.086,281.554,385.776,171.482,42.296,158.099
C05140=1039.079,281.306,385.807,171.479,42.294,158.099
C05141=1039.072,281.058,385.839,171.475,42.293,158.098
C05142=1039.065,280.810,385.870,171.471,42.291,158.097
C05143=1039.059,280.563,385.901,171.468,42.290,158.097
C05144=1039.052,280.315,385.932,171.465,42.288,158.096
C05145=1039.046,280.067,385.963,171.461,42.286,158.096
C05146=1039.039,279.819,385.994,171.458,42.285,158.095
C05147=1039.032,279.571,386.025,171.454,42.283,158.094
C05148=1039.025,279.323,386.057,171.451,42.281,158.094
C05149=1039.018,279.075,386.088,171.447,42.280,158.093
C05150=1039.012,278.827,386.120,171.444,42.279,158.093
C05151=1039.005,278.579,386.150,171.440,42.277,158.092
C05152=1038.999,278.331,386.182,171.437,42.275,158.092
C05153=1038.992,278.083,386.213,171.434,42.274,158.091
C05154=1038.985,277.835,386.245,171.430,42.272,158.091
C05155=1038.976,277.516,386.285,171.426,42.270,158.090
C05156=1038.968,277.196,386.324,171.422,42.269,158.089
C05157=1038.959,276.877,386.364,171.418,42.267,158.088
C05158=1038.950,276.558,386.404,171.413,42.265,158.088
C05159=1038.944,276.310,386.435,171.409,42.263,158.087
C05160=1038.937,276.062,386.466,171.407,42.261,158.087
C05161=1038.930,275.814,386.497,171.403,42.260,158.086
C05162=1038.923,275.566,386.528,171.399,42.258,158.085
C05163=1038.917,275.318,386.558,171.396,42.257,158.085
C05164=1038.910,275.071,386.589,171.393,42.256,158.084
C05165=1038.903,274.822,386.620,171.389,42.254,158.084
C05166=1038.897,274.574,386.651,171.386,42.252,158.083
C05167=1038.890,274.326,386.682,171.383,42.251,158.083
C05168=1038.883,274.078,386.713,171.379,42.249,158.082
C05169=1038.877,273.830,386.743,171.376,42.248,158.082
C05170=1038.870,273.582,386.775,171.372,42.247,158.081
C05171=1038.863,273.334,386.805,171.370,42.245,158.081
C05172=1038.856,273.086,386.836,171.366,42.244,158.080
C05173=1038.849,272.838,386.866,171.362,42.242,158.079
C05174=1038.843,272.590,386.897,171.360,42.241,158.079
C05175=1038.837,272.342,386.928,171.356,42.239,158.078
C05176=1038.829,272.094,386.958,171.353,42.238,158.078
C05177=1038.823,271.846,386.989,171.350,42.236,158.077
C05178=1038.817,271.598,387.020,171.346,42.234,158.077
C05179=1038.810,271.350,387.050,171.342,42.233,158.076
C05180=1038.803,271.102,387.081,171.340,42.231,158.076
C05181=1038.796,270.854,387.112,171.336,42.230,158.075
C05182=1038.789,270.606,387.142,171.333,42.229,158.075
C05183=1038.783,270.358,387.172,171.330,42.227,158.074
C05184=1038.776,270.110,387.204,171.326,42.226,158.073
C05185=1038.769,269.862,387.234,171.324,42.224,158.073
C05186=1038.763,269.613,387.264,171.320,42.223,158.072
C05187=1038.756,269.366,387.294,171.317,42.222,158.072
C05188=1038.750,269.117,387.325,171.314,42.220,158.071
C05189=1038.742,268.870,387.356,171.310,42.219,158.071
C05190=1038.736,268.622,387.386,171.307,42.217,158.070
C05191=1038.729,268.374,387.416,171.304,42.216,158.070
C05192=1038.722,268.126,387.446,171.301,42.215,158.069
C05193=1038.716,267.877,387.477,171.297,42.214,158.069
C05194=1038.709,267.630,387.507,171.295,42.212,158.068
C05195=1038.703,267.381,387.538,171.291,42.211,158.068
C05196=1038.695,267.133,387.568,171.288,42.209,158.067
C05197=1038.690,266.885,387.598,171.285,42.208,158.067
C05198=1038.682,266.637,387.628,171.281,42.206,158.066
C05199=1038.675,266.389,387.659,171.278,42.205,158.066
C05200=1038.668,266.142,387.689,171.275,42.203,158.065
C05201=1038.662,265.893,387.719,171.272,42.202,158.065
C05202=1038.655,265.644,387.749,171.269,42.200,158.064
C05203=1038.649,265.397,387.779,171.265,42.200,158.064
C05204=1038.642,265.148,387.809,171.263,42.198,158.063
C05205=1038.635,264.900,387.839,171.259,42.197,158.063
C05206=1038.629,264.653,387.869,171.256,42.195,158.062
C05207=1038.622,264.404,387.900,171.253,42.194,158.062
C05208=1038.616,264.157,387.930,171.250,42.192,158.061
C05209=1038.608,263.908,387.960,171.247,42.191,158.061
C05210=1038.602,263.660,387.991,171.243,42.190,158.060
C05211=1038.593,263.345,388.028,171.239,42.188,158.059
C05212=1038.585,263.031,388.067,171.236,42.186,158.059
C05213=1038.576,262.716,388.104,171.232,42.185,158.058
C05214=1038.568,262.401,388.142,171.227,42.183,158.058
C05215=1038.562,262.153,388.172,171.225,42.181,158.057
C05216=1038.555,261.905,388.202,171.221,42.180,158.057
C05217=1038.548,261.658,388.232,171.219,42.179,158.056
C05218=1038.541,261.409,388.261,171.215,42.178,158.056
C05219=1038.534,261.160,388.292,171.212,42.176,158.055
C05220=1038.527,260.913,388.321,171.209,42.175,158.055
C05221=1038.521,260.664,388.351,171.206,42.174,158.054
C05222=1038.514,260.417,388.381,171.203,42.172,158.054
C05223=1038.507,260.168,388.411,171.199,42.172,158.053
C05224=1038.500,259.920,388.440,171.197,42.170,158.053
C05225=1038.493,259.672,388.470,171.193,42.169,158.052
C05226=1038.487,259.423,388.499,171.191,42.168,158.052
C05227=1038.480,259.176,388.529,171.187,42.166,158.051
C05228=1038.473,258.927,388.558,171.184,42.165,158.051
C05229=1038.466,258.680,388.588,171.181,42.164,158.050
C05230=1038.459,258.431,388.617,171.178,42.162,158.050
C05231=1038.452,258.183,388.647,171.175,42.161,158.049
C05232=1038.445,257.935,388.677,171.172,42.160,158.049
C05233=1038.439,257.686,388.706,171.169,42.159,158.048
C05234=1038.432,257.438,388.735,171.166,42.157,158.048
C05235=1038.425,257.190,388.765,171.163,42.156,158.048
C05236=1038.419,256.942,388.794,171.160,42.155,158.047
C05237=1038.412,256.694,388.825,171.157,42.153,158.047
C05238=1038.405,256.445,388.854,171.154,42.152,158.046
C05239=1038.398,256.198,388.883,171.151,42.151,158.046
C05240=1038.391,255.949,388.912,171.148,42.149,158.045
C05241=1038.384,255.701,388.942,171.145,42.149,158.045
C05242=1038.378,255.453,388.971,171.142,42.147,158.044
C05243=1038.371,255.204,389.001,171.138,42.146,158.044
C05244=1038.365,254.957,389.030,171.136,42.145,158.043
C05245=1038.358,254.709,389.060,171.132,42.143,158.043
C05246=1038.351,254.460,389.089,171.130,42.142,158.042
C05247=1038.345,254.212,389.119,171.126,42.141,158.042
C05248=1038.337,253.964,389.147,171.124,42.140,158.041
C05249=1038.331,253.716,389.177,171.120,42.139,158.041
C05250=1038.324,253.467,389.207,171.118,42.137,158.041
C05251=1038.318,253.219,389.236,171.114,42.136,158.040
C05252=1038.311,252.971,389.265,171.112,42.135,158.040
C05253=1038.304,252.723,389.295,171.109,42.133,158.039
C05254=1038.298,252.475,389.324,171.106,42.132,158.039
C05255=1038.291,252.226,389.353,171.103,42.131,158.038
C05256=1038.284,251.978,389.382,171.100,42.130,158.038
C05257=1038.278,251.731,389.412,171.097,42.129,158.037
C05258=1038.271,251.482,389.441,171.094,42.127,158.037
C05259=1038.264,251.234,389.470,171.091,42.126,158.036
C05260=1038.258,250.986,389.499,171.089,42.125,158.036
C05261=1038.251,250.737,389.528,171.085,42.123,158.035
C05262=1038.245,250.489,389.557,171.082,42.122,158.035
C05263=1038.238,250.241,389.587,171.079,42.121,158.034
C05264=1038.231,249.993,389.616,171.076,42.119,158.034
C05265=1038.225,249.744,389.645,171.074,42.118,158.034
C05266=1038.218,249.496,389.674,171.070,42.117,158.033
C05267=1038.210,249.180,389.712,171.067,42.116,158.033
C05268=1038.201,248.865,389.748,171.063,42.114,158.032
C05269=1038.193,248.548,389.785,171.059,42.112,158.031
C05270=1038.185,248.231,389.823,171.056,42.111,158.031
C05271=1038.179,247.983,389.852,171.053,42.109,158.030
C05272=1038.172,247.735,389.881,171.050,42.108,158.030
C05273=1038.165,247.487,389.909,171.047,42.107,158.029
C05274=1038.159,247.238,389.939,171.044,42.105,158.029
C05275=1038.152,246.990,389.968,171.041,42.105,158.029
C05276=1038.146,246.742,389.997,171.038,42.103,158.028
C05277=1038.140,246.494,390.026,171.036,42.101,158.028
C05278=1038.133,246.245,390.055,171.032,42.101,158.027
C05279=1038.126,245.997,390.084,171.030,42.099,158.027
C05280=1038.120,245.749,390.113,171.027,42.098,158.026
C05281=1038.113,245.501,390.142,171.025,42.097,158.026
C05282=1038.107,245.253,390.171,171.021,42.095,158.025
C05283=1038.100,245.004,390.200,171.019,42.094,158.025
C05284=1038.093,244.756,390.229,171.016,42.093,158.024
C05285=1038.087,244.508,390.258,171.013,42.092,158.024
C05286=1038.080,244.260,390.286,171.010,42.090,158.023
C05287=1038.074,244.011,390.315,171.008,42.089,158.023
C05288=1038.067,243.763,390.344,171.004,42.088,158.023
C05289=1038.060,243.515,390.372,171.002,42.087,158.022
C05290=1038.054,243.267,390.401,170.999,42.085,158.022
C05291=1038.047,243.019,390.430,170.996,42.085,158.021
C05292=1038.041,242.770,390.459,170.993,42.083,158.021
C05293=1038.034,242.522,390.487,170.991,42.082,158.020
C05294=1038.027,242.274,390.516,170.987,42.081,158.020
C05295=1038.021,242.025,390.545,170.985,42.080,158.020
C05296=1038.014,241.777,390.573,170.982,42.078,158.019
C05297=1038.008,241.529,390.602,170.979,42.077,158.019
C05298=1038.001,241.280,390.631,170.976,42.076,158.018
C05299=1037.995,241.032,390.659,170.974,42.075,158.018
C05300=1037.988,240.784,390.687,170.971,42.073,158.017
C05301=1037.981,240.536,390.716,170.968,42.073,158.017
C05302=1037.975,240.287,390.744,170.965,42.072,158.017
C05303=1037.968,240.039,390.773,170.963,42.070,158.016
C05304=1037.961,239.790,390.801,170.959,42.069,158.016
C05305=1037.954,239.542,390.830,170.957,42.068,158.015
C05306=1037.947,239.294,390.858,170.954,42.067,158.015
C05307=1037.941,239.046,390.887,170.952,42.066,158.014
C05308=1037.934,238.798,390.915,170.948,42.064,158.014
C05309=1037.928,238.549,390.943,170.946,42.063,158.014
C05310=1037.921,238.301,390.972,170.943,42.062,158.013
C05311=1037.914,238.052,391.000,170.940,42.061,158.013
C05312=1037.907,237.804,391.028,170.938,42.060,158.012
C05313=1037.901,237.555,391.057,170.935,42.059,158.012
C05314=1037.894,237.308,391.085,170.933,42.058,158.011
C05315=1037.887,237.059,391.113,170.929,42.057,158.011
C05316=1037.881,236.811,391.141,170.927,42.055,158.011
C05317=1037.874,236.563,391.170,170.924,42.054,158.010
C05318=1037.868,236.314,391.197,170.922,42.053,158.010
C05319=1037.861,236.066,391.226,170.918,42.052,158.009
C05320=1037.854,235.817,391.254,170.916,42.051,158.009
C05321=1037.848,235.568,391.282,170.913,42.049,158.008
C05322=1037.841,235.321,391.311,170.911,42.049,158.008
C05323=1037.832,234.999,391.347,170.907,42.047,158.008
C05324=1037.824,234.677,391.383,170.904,42.046,158.007
C05325=1037.815,234.355,391.420,170.900,42.044,158.007
C05326=1037.807,234.033,391.456,170.896,42.043,158.006
C05327=1037.800,233.785,391.484,170.894,42.042,158.006
C05328=1037.793,233.537,391.512,170.891,42.040,158.005
C05329=1037.786,233.288,391.541,170.888,42.039,158.005
C05330=1037.780,233.039,391.569,170.885,42.038,158.004
C05331=1037.773,232.791,391.597,170.883,42.037,158.004
C05332=1037.766,232.542,391.624,170.881,42.036,158.004
C05333=1037.759,232.295,391.653,170.878,42.034,158.003
C05334=1037.753,232.046,391.681,170.875,42.034,158.003
C05335=1037.747,231.797,391.709,170.872,42.033,158.002
C05336=1037.740,231.549,391.737,170.870,42.031,158.002
C05337=1037.733,231.301,391.765,170.867,42.030,158.001
C05338=1037.726,231.053,391.793,170.865,42.029,158.001
C05339=1037.720,230.804,391.821,170.862,42.028,158.001
C05340=1037.714,230.556,391.848,170.859,42.027,158.000
C05341=1037.707,230.308,391.876,170.857,42.026,158.000
C05342=1037.701,230.059,391.904,170.854,42.024,157.999
C05343=1037.694,229.811,391.932,170.852,42.023,157.999
C05344=1037.688,229.562,391.959,170.849,42.022,157.999
C05345=1037.681,229.315,391.988,170.847,42.021,157.998
C05346=1037.674,229.066,392.016,170.843,42.020,157.998
C05347=1037.667,228.818,392.043,170.841,42.019,157.997
C05348=1037.661,228.569,392.071,170.838,42.018,157.997
C05349=1037.654,228.321,392.099,170.836,42.017,157.997
C05350=1037.647,228.072,392.127,170.833,42.016,157.996
C05351=1037.641,227.824,392.154,170.831,42.015,157.996
C05352=1037.634,227.575,392.182,170.828,42.014,157.995
C05353=1037.627,227.327,392.210,170.825,42.012,157.995
C05354=1037.620,227.079,392.237,170.823,42.011,157.995
C05355=1037.613,226.830,392.265,170.820,42.010,157.994
C05356=1037.606,226.582,392.292,170.818,42.009,157.994
C05357=1037.600,226.333,392.319,170.815,42.008,157.994
C05358=1037.593,226.085,392.347,170.812,42.007,157.993
C05359=1037.587,225.836,392.375,170.809,42.006,157.993
C05360=1037.580,225.588,392.403,170.807,42.005,157.992
C05361=1037.573,225.340,392.429,170.805,42.004,157.992
C05362=1037.567,225.092,392.457,170.802,42.003,157.991
C05363=1037.560,224.843,392.485,170.800,42.002,157.991
C05364=1037.553,224.595,392.512,170.797,42.001,157.991
C05365=1037.547,224.346,392.539,170.795,42.000,157.990
C05366=1037.540,224.097,392.567,170.791,41.999,157.990
C05367=1037.533,223.849,392.594,170.789,41.997,157.989
C05368=1037.526,223.601,392.622,170.786,41.996,157.989
C05369=1037.519,223.352,392.650,170.784,41.995,157.989
C05370=1037.513,223.105,392.677,170.782,41.994,157.988
C05371=1037.507,222.856,392.704,170.779,41.993,157.988
C05372=1037.500,222.607,392.732,170.777,41.992,157.988
C05373=1037.493,222.359,392.759,170.774,41.991,157.987
C05374=1037.486,222.111,392.787,170.772,41.990,157.987
C05375=1037.480,221.861,392.814,170.769,41.988,157.986
C05376=1037.474,221.614,392.841,170.766,41.988,157.986
C05377=1037.467,221.365,392.869,170.763,41.987,157.986
C05378=1037.460,221.117,392.897,170.761,41.986,157.985
C05379=1037.452,220.787,392.932,170.758,41.984,157.985
C05380=1037.443,220.458,392.968,170.755,41.983,157.984
C05381=1037.434,220.128,393.005,170.751,41.981,157.984
C05382=1037.425,219.799,393.041,170.748,41.980,157.983
C05383=1037.418,219.550,393.069,170.745,41.979,157.983
C05384=1037.411,219.302,393.095,170.743,41.978,157.982
C05385=1037.405,219.054,393.122,170.740,41.977,157.982
C05386=1037.398,218.805,393.149,170.738,41.975,157.982
C05387=1037.391,218.557,393.177,170.735,41.974,157.981
C05388=1037.384,218.308,393.203,170.733,41.973,157.981
C05389=1037.378,218.060,393.231,170.731,41.973,157.981
C05390=1037.370,217.811,393.258,170.728,41.972,157.980
C05391=1037.364,217.563,393.284,170.726,41.971,157.980
C05392=1037.358,217.315,393.312,170.724,41.970,157.980
C05393=1037.351,217.066,393.339,170.721,41.968,157.979
C05394=1037.344,216.817,393.366,170.719,41.967,157.979
C05395=1037.338,216.569,393.392,170.716,41.966,157.978
C05396=1037.331,216.320,393.419,170.714,41.965,157.978
C05397=1037.324,216.072,393.447,170.711,41.964,157.978
C05398=1037.317,215.823,393.474,170.708,41.963,157.977
C05399=1037.311,215.576,393.500,170.706,41.962,157.977
C05400=1037.304,215.327,393.527,170.703,41.961,157.976
C05401=1037.297,215.079,393.554,170.701,41.960,157.976
C05402=1037.290,214.829,393.582,170.698,41.959,157.976
C05403=1037.284,214.582,393.609,170.696,41.958,157.975
C05404=1037.277,214.333,393.635,170.693,41.957,157.975
C05405=1037.271,214.084,393.662,170.691,41.956,157.975
C05406=1037.264,213.837,393.689,170.689,41.955,157.974
C05407=1037.258,213.587,393.716,170.686,41.953,157.974
C05408=1037.250,213.339,393.743,170.684,41.953,157.973
C05409=1037.244,213.091,393.770,170.681,41.952,157.973
C05410=1037.237,212.842,393.796,170.679,41.951,157.973
C05411=1037.231,212.593,393.823,170.676,41.950,157.972
C05412=1037.223,212.345,393.850,170.674,41.949,157.972
C05413=1037.218,212.097,393.877,170.672,41.947,157.972
C05414=1037.211,211.848,393.904,170.670,41.946,157.971
C05415=1037.205,211.600,393.931,170.668,41.945,157.971
C05416=1037.197,211.351,393.957,170.665,41.944,157.970
C05417=1037.191,211.102,393.984,170.663,41.943,157.970
C05418=1037.185,210.854,394.010,170.660,41.942,157.970
C05419=1037.177,210.606,394.037,170.658,41.941,157.969
C05420=1037.171,210.357,394.065,170.656,41.940,157.969
C05421=1037.164,210.109,394.091,170.653,41.939,157.969
C05422=1037.157,209.860,394.117,170.651,41.938,157.968
C05423=1037.151,209.611,394.144,170.648,41.937,157.968
C05424=1037.144,209.364,394.171,170.646,41.936,157.968
C05425=1037.138,209.115,394.198,170.644,41.935,157.967
C05426=1037.130,208.866,394.224,170.641,41.934,157.967
C05427=1037.124,208.618,394.250,170.639,41.933,157.966
C05428=1037.117,208.369,394.277,170.636,41.932,157.966
C05429=1037.110,208.120,394.304,170.634,41.931,157.966
C05430=1037.104,207.872,394.330,170.632,41.930,157.965
C05431=1037.097,207.623,394.356,170.629,41.928,157.965
C05432=1037.090,207.376,394.383,170.627,41.927,157.965
C05433=1037.084,207.127,394.410,170.624,41.926,157.964
C05434=1037.076,206.878,394.436,170.622,41.925,157.964
C05435=1037.068,206.555,394.470,170.619,41.924,157.963
C05436=1037.059,206.231,394.504,170.616,41.923,157.963
C05437=1037.050,205.907,394.539,170.613,41.921,157.962
C05438=1037.042,205.583,394.574,170.610,41.921,157.962
C05439=1037.015,204.533,394.679,170.301,41.816,157.921
C05440=1037.009,204.284,394.705,170.298,41.816,157.921
C05441=1037.003,204.035,394.730,170.295,41.816,157.921
C05442=1036.997,203.787,394.755,170.292,41.815,157.921
C05443=1036.991,203.537,394.780,170.288,41.815,157.920
C05444=1036.985,203.289,394.805,170.285,41.815,157.920
C05445=1036.979,203.041,394.830,170.282,41.814,157.920
C05446=1036.972,202.792,394.855,170.279,41.814,157.920
C05447=1036.966,202.543,394.880,170.275,41.814,157.919
C05448=1036.960,202.295,394.905,170.272,41.813,157.919
C05449=1036.954,202.046,394.930,170.269,41.813,157.919
C05450=1036.948,201.797,394.956,170.266,41.813,157.919
C05451=1036.942,201.549,394.980,170.262,41.813,157.918
C05452=1036.936,201.300,395.005,170.259,41.813,157.918
C05453=1036.930,201.051,395.031,170.256,41.812,157.918
C05454=1036.924,200.802,395.055,170.253,41.812,157.918
C05455=1036.917,200.554,395.080,170.250,41.812,157.917
C05456=1036.911,200.305,395.105,170.246,41.812,157.917
C05457=1036.905,200.057,395.129,170.243,41.812,157.917
C05458=1036.899,199.808,395.154,170.241,41.811,157.917
